		CASE etDiagExtModuleController OF
			TPL.ET_DiagExt.DeactivatingSubModules : 
				stMachineInterface.q_udiDiagExt	:= ET_DiagExt.DeactivatingSubModules;
				stMachineInterface.q_sDiagExt		:= FC_EtDiagExtToString(i_etDiagExt := ET_DiagExt.DeactivatingSubModules);
			TPL.ET_DiagExt.Disabled : 
				stMachineInterface.q_udiDiagExt	:= ET_DiagExt.Disabled;
				stMachineInterface.q_sDiagExt		:= FC_EtDiagExtToString(i_etDiagExt := ET_DiagExt.Disabled);
			TPL.ET_DiagExt.ExecuteStep : 
				stMachineInterface.q_udiDiagExt	:= ET_DiagExt.ExecuteStep;
				stMachineInterface.q_sDiagExt		:= FC_EtDiagExtToString(i_etDiagExt := ET_DiagExt.ExecuteStep);
			TPL.ET_DiagExt.Initializing : 
				stMachineInterface.q_udiDiagExt	:= ET_DiagExt.Initializing;
				stMachineInterface.q_sDiagExt		:= FC_EtDiagExtToString(i_etDiagExt := ET_DiagExt.Initializing);
			TPL.ET_DiagExt.WaitAtNegativeStep : 
				stMachineInterface.q_udiDiagExt	:= ET_DiagExt.WaitAtNegativeStep;
				stMachineInterface.q_sDiagExt		:= FC_EtDiagExtToString(i_etDiagExt := ET_DiagExt.WaitAtNegativeStep);
			TPL.ET_DiagExt.WaitCmdsDone : 
				stMachineInterface.q_udiDiagExt	:= ET_DiagExt.WaitCmdsDone;
				stMachineInterface.q_sDiagExt		:= FC_EtDiagExtToString(i_etDiagExt := ET_DiagExt.WaitCmdsDone);
			TPL.ET_DiagExt.WaitForCmd : 
				stMachineInterface.q_udiDiagExt	:= ET_DiagExt.WaitForCmd;
				stMachineInterface.q_sDiagExt		:= FC_EtDiagExtToString(i_etDiagExt := ET_DiagExt.WaitForCmd);
			ELSE
				stMachineInterface.q_etDiag		:= GD. ET_Diag.UnexpectedProgramBehavior;
				stMachineInterface.q_udiDiagExt	:= ET_DiagExt.UnknownStateModuleController;
				stMachineInterface.q_sDiagExt		:= FC_EtDiagExtToString(i_etDiagExt := ET_DiagExt.UnknownStateModuleController);
		END_CASE
	ELSE
		stMachineInterface.q_etDiag		:= GD.ET_Diag.DiagActive;
		stMachineInterface.q_udiDiagExt	:= ET_DiagExt.ModuleControllerException;
		stMachineInterface.q_sDiagExt		:= FC_EtDiagExtToString(i_etDiagExt := ET_DiagExt.ModuleControllerException);
		stMachineInterface.q_sMsg			:= PDL.FC_MultiConcat(	i_sString1 := GD.FC_EtDiagToString(i_etDiag := etDiagModuleController), 
																			i_sString2 := ' - ',
																			i_sString3 := TPL.FC_EtDiagExtToString(i_etDiagExt := etDiagExtModuleController), 
																			i_sString4 := '');
	END_IF
END_IF
(* End of system generated code, only to be changed by experienced programmers *)
END_ACTION

ACTION PrepStep_Action:
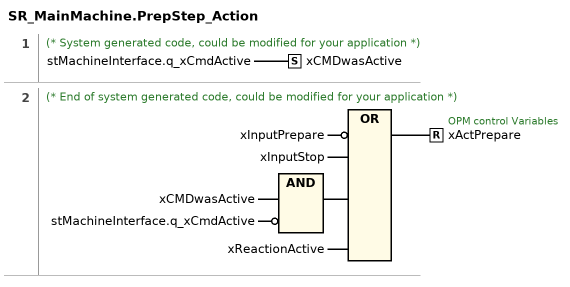
// NETWORK 1
// (* System generated code, could be modified for your application *)
xCMDwasActive S= stMachineInterface.q_xCmdActive;

// NETWORK 2
// (* End of system generated code, could be modified for your application *)
//   xActPrepare: OPM control Variables
xActPrepare R= NOT xInputPrepare OR xInputStop OR xCMDwasActive AND NOT stMachineInterface.q_xCmdActive OR xReactionActive;
END_ACTION

ACTION PrepStep_Entry:
(* System generated code, could be modified for your application *)
	xCMDwasActive:=FALSE;
	stMachineInterface.iq_diCmd	:= ET_Cmd.Prepare;
(* End of system generated code, could be modified for your application *)
END_ACTION

ACTION PrepStop_Action:
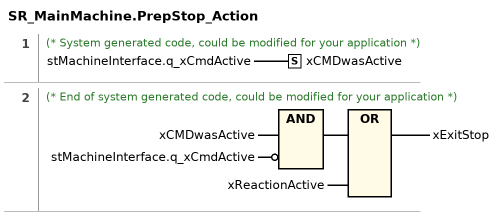
// NETWORK 1
// (* System generated code, could be modified for your application *)
xCMDwasActive S= stMachineInterface.q_xCmdActive;

// NETWORK 2
// (* End of system generated code, could be modified for your application *)
xExitStop := xCMDwasActive AND NOT stMachineInterface.q_xCmdActive OR xReactionActive;
END_ACTION

ACTION PrepStop_Entry:
(* System generated code, could be modified for your application *)
	xCMDwasActive:=FALSE;
	IF	xReactionActive	THEN
		;
	ELSIF stMachineInterface.q_xCmdDone AND NOT stMachineInterface.q_xCmdActive THEN
		stMachineInterface.iq_diCmd	:= ET_Cmd.Stop;
	ELSE
		stMachineInterface.iq_diCmd	:= ET_Cmd.Abort;
	END_IF
(* End of system generated code, could be modified for your application *)
END_ACTION

ACTION StopBrake_Action:
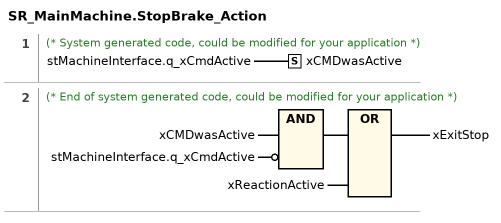
// NETWORK 1
// (* System generated code, could be modified for your application *)
xCMDwasActive S= stMachineInterface.q_xCmdActive;

// NETWORK 2
// (* End of system generated code, could be modified for your application *)
xExitStop := xCMDwasActive AND NOT stMachineInterface.q_xCmdActive OR xReactionActive;
END_ACTION

ACTION StopBrake_Entry:
(* System generated code, could be modified for your application *)
	xCMDwasActive:=FALSE;
	IF	xReactionActive	THEN
		stMachineInterface.iq_diCmd	:= ET_Cmd.Stop;
	ELSIF stMachineInterface.q_xCmdDone AND NOT stMachineInterface.q_xCmdActive THEN
		stMachineInterface.iq_diCmd	:= ET_Cmd.Stop;
	ELSE
		stMachineInterface.iq_diCmd	:= ET_Cmd.Abort;
	END_IF
(* End of system generated code, could be modified for your application *)
END_ACTION

ACTION StopJog_Action:
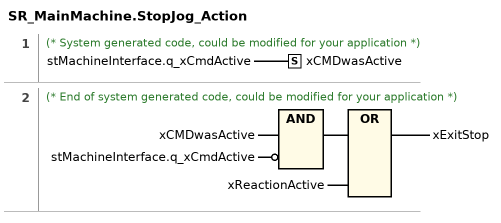
// NETWORK 1
// (* System generated code, could be modified for your application *)
xCMDwasActive S= stMachineInterface.q_xCmdActive;

// NETWORK 2
// (* End of system generated code, could be modified for your application *)
xExitStop := xCMDwasActive AND NOT stMachineInterface.q_xCmdActive OR xReactionActive;
END_ACTION

ACTION StopJog_Entry:
(* System generated code, could be modified for your application *)
	xCMDwasActive:=FALSE;
	IF	xReactionActive	THEN
		;
	ELSIF stMachineInterface.q_xCmdDone AND NOT stMachineInterface.q_xCmdActive THEN
		stMachineInterface.iq_diCmd	:= ET_Cmd.HoldJM;
	ELSE
		stMachineInterface.iq_diCmd	:= ET_Cmd.Abort;
	END_IF
(* End of system generated code, could be modified for your application *)
END_ACTION

ACTION StopMan_Action:
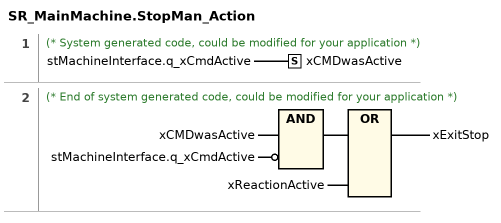
// NETWORK 1
// (* System generated code, could be modified for your application *)
xCMDwasActive S= stMachineInterface.q_xCmdActive;

// NETWORK 2
// (* End of system generated code, could be modified for your application *)
xExitStop := xCMDwasActive AND NOT stMachineInterface.q_xCmdActive OR xReactionActive;
END_ACTION

ACTION StopMan_Entry:
(* System generated code, could be modified for your application *)
	xCMDwasActive:=FALSE;
	IF	xReactionActive	THEN
		;
	ELSIF stMachineInterface.q_xCmdDone AND NOT stMachineInterface.q_xCmdActive THEN
		stMachineInterface.iq_diCmd	:= ET_Cmd.Stop;
	ELSE
		stMachineInterface.iq_diCmd	:= ET_Cmd.Abort;
	END_IF
(* End of system generated code, could be modified for your application *)
END_ACTION

ACTION SubModules_Action:
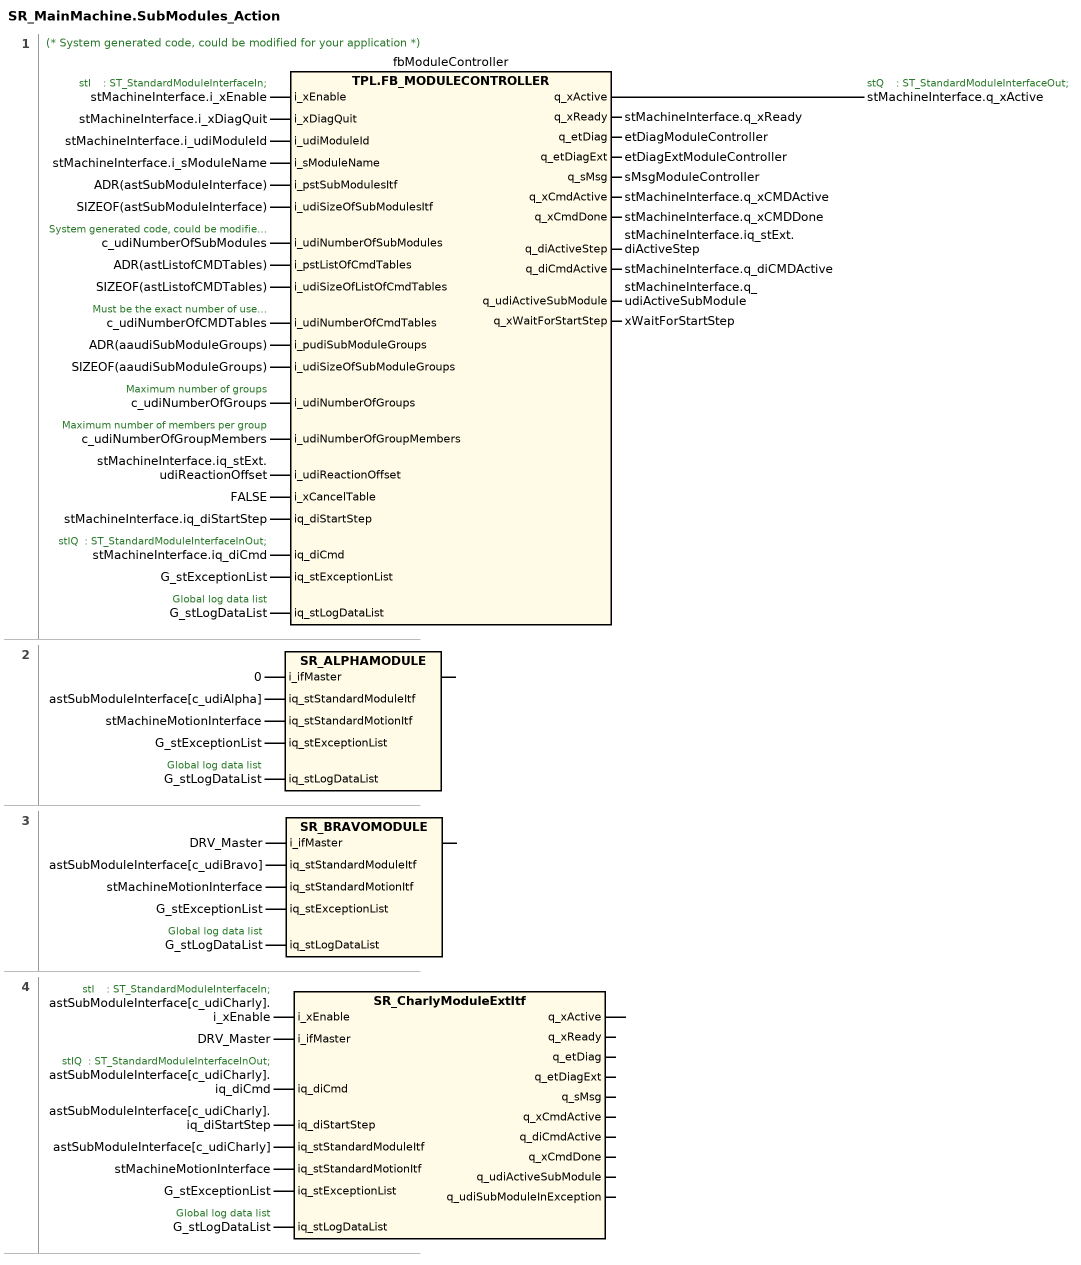
// NETWORK 1
// (* System generated code, could be modified for your application *)
//   fbModuleController: Main ModuleController
//   stMachineInterface.i_xEnable: stI : ST_StandardModuleInterfaceIn;
//   c_udiNumberOfSubModules: System generated code, could be modified for your application
//   c_udiNumberOfCMDTables: Must be the exact number of used CMDTables!
//   c_udiNumberOfGroups: Maximum number of groups
//   c_udiNumberOfGroupMembers: Maximum number of members per group
//   stMachineInterface.iq_diCmd: stIQ : ST_StandardModuleInterfaceInOut;
//   G_stLogDataList: Global log data list
//   stMachineInterface.q_xActive: stQ : ST_StandardModuleInterfaceOut;
fbModuleController(
    i_xEnable := stMachineInterface.i_xEnable,
    i_xDiagQuit := stMachineInterface.i_xDiagQuit,
    i_udiModuleId := stMachineInterface.i_udiModuleId,
    i_sModuleName := stMachineInterface.i_sModuleName,
    i_pstSubModulesItf := ADR(astSubModuleInterface),
    i_udiSizeOfSubModulesItf := SIZEOF(astSubModuleInterface),
    i_udiNumberOfSubModules := c_udiNumberOfSubModules,
    i_pstListOfCmdTables := ADR(astListofCMDTables),
    i_udiSizeOfListOfCmdTables := SIZEOF(astListofCMDTables),
    i_udiNumberOfCmdTables := c_udiNumberOfCMDTables,
    i_pudiSubModuleGroups := ADR(aaudiSubModuleGroups),
    i_udiSizeOfSubModuleGroups := SIZEOF(aaudiSubModuleGroups),
    i_udiNumberOfGroups := c_udiNumberOfGroups,
    i_udiNumberOfGroupMembers := c_udiNumberOfGroupMembers,
    i_udiReactionOffset := stMachineInterface.iq_stExt.udiReactionOffset,
    i_xCancelTable := FALSE,
    iq_diStartStep := stMachineInterface.iq_diStartStep,
    iq_diCmd := stMachineInterface.iq_diCmd,
    iq_stExceptionList := G_stExceptionList,
    iq_stLogDataList := G_stLogDataList,
    q_xReady => stMachineInterface.q_xReady,
    q_etDiag => etDiagModuleController,
    q_etDiagExt => etDiagExtModuleController,
    q_sMsg => sMsgModuleController,
    q_xCmdActive => stMachineInterface.q_xCMDActive,
    q_xCmdDone => stMachineInterface.q_xCMDDone,
    q_diActiveStep => stMachineInterface.iq_stExt.diActiveStep,
    q_diCmdActive => stMachineInterface.q_diCMDActive,
    q_udiActiveSubModule => stMachineInterface.q_udiActiveSubModule,
    q_xWaitForStartStep => xWaitForStartStep); // TPL.FB_MODULECONTROLLER
stMachineInterface.q_xActive := fbModuleController.q_xActive;

// NETWORK 2
//   G_stLogDataList: Global log data list
SR_ALPHAMODULE(i_ifMaster := 0, iq_stStandardModuleItf := astSubModuleInterface[c_udiAlpha], iq_stStandardMotionItf := stMachineMotionInterface, iq_stExceptionList := G_stExceptionList, iq_stLogDataList := G_stLogDataList);

// NETWORK 3
//   G_stLogDataList: Global log data list
SR_BRAVOMODULE(i_ifMaster := DRV_Master, iq_stStandardModuleItf := astSubModuleInterface[c_udiBravo], iq_stStandardMotionItf := stMachineMotionInterface, iq_stExceptionList := G_stExceptionList, iq_stLogDataList := G_stLogDataList);

// NETWORK 4
//   astSubModuleInterface[c_udiCharly].i_xEnable: stI : ST_StandardModuleInterfaceIn;
//   astSubModuleInterface[c_udiCharly].iq_diCmd: stIQ : ST_StandardModuleInterfaceInOut;
//   G_stLogDataList: Global log data list
SR_CharlyModuleExtItf(i_xEnable := astSubModuleInterface[c_udiCharly].i_xEnable, i_ifMaster := DRV_Master, iq_diCmd := astSubModuleInterface[c_udiCharly].iq_diCmd, iq_diStartStep := astSubModuleInterface[c_udiCharly].iq_diStartStep, iq_stStandardModuleItf := astSubModuleInterface[c_udiCharly], iq_stStandardMotionItf := stMachineMotionInterface, iq_stExceptionList := G_stExceptionList, iq_stLogDataList := G_stLogDataList);

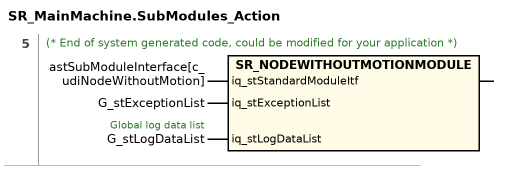
// NETWORK 5
// (* End of system generated code, could be modified for your application *)
//   G_stLogDataList: Global log data list
SR_NODEWITHOUTMOTIONMODULE(iq_stStandardModuleItf := astSubModuleInterface[c_udiNodeWithoutMotion], iq_stExceptionList := G_stExceptionList, iq_stLogDataList := G_stLogDataList);
END_ACTION

ACTION UpdateStructs:
(* System generated code, do not change without consulting 'Schneider Electric Automation GmbH' - otherwise you risk instability!!!*)
fbDetectOnlineChange(	i_xEnable	:= TRUE, 
						i_xDetect	:= TRUE, 
						q_xActive	=> xDetectOnlineChangeActive, 
						q_xReady	=> xDetectOnlineChangeReady, 
						q_etDiag	=> etDetectOnlineChangeDiag, 
						q_etDiagExt	=> etDetectOnlineChangeDiagExt, 
						q_sMsg		=> sDetectOnlineChangeMsg, 
						q_xChange	=> );
						
IF(NOT fbDetectOnlineChange.q_xChange) THEN
	RETURN;
END_IF

stMachineInterface.iq_stExt.udiNumberOfSubModules 		:= c_udiNumberOfSubModules;
stMachineInterface.iq_stExt.dwSubModulesItf		 		:= ADR(astSubModuleInterface);
stMachineInterface.iq_stExt.pdwSubModulesAddItf			:= ADR(adwSubModuleAddInterfaces);
stMachineInterface.iq_stExt.pstListofCMDTables			:= ADR(astListOfCMDTables);
stMachineInterface.iq_stExt.udiNumberOfCmdTables		:= c_udiNumberOfCMDTables;
(* End of system generated code, do not change without consulting 'Schneider Electric Automation GmbH' - otherwise you risk instability!!!*)

(* System generated code, could be modified for your application *)

xUpdateStructsException := FALSE;

(*****************************************************************************************************************************************************)
(* Update CmdTable - Prepare *)

TPL.FC_UpdateCmdTableListElement(	i_pstListofCMDTables	:= ADR(astListofCMDTables),
									i_udiNumberOfCmdTables	:= c_udiNumberOfCMDTables,
									i_diCMD					:= ET_Cmd.Prepare,
									i_pstCMDTable			:= ADR(astPrepareTable),
									q_etDiag				=> etDiag,
									q_etDiagExt				=> etDiagExtTPL);
									
IF etDiag <> GD.ET_Diag.Ok AND NOT xUpdateStructsException THEN
	xUpdateStructsException := TRUE;
	
	stUpdateStructsException.sMsg := PDL.FC_MultiConcat(i_sString1 := 'Update CmdTable: Prepare - ', 
														i_sString2 := GD.FC_EtDiagToString(i_etDiag := etDiag), 
														i_sString3 := ' - ', 
														i_sString4 := TPL.FC_EtDiagExtToString(i_etDiagExt := etDiagExtTPL));
END_IF										

(*****************************************************************************************************************************************************)
(* Update CmdTable - Auto *)

TPL.FC_UpdateCmdTableListElement(	i_pstListofCMDTables	:= ADR(astListofCMDTables),
									i_udiNumberOfCMDTables	:= c_udiNumberOfCMDTables,
									i_diCMD					:= ET_Cmd.Auto,
									i_pstCMDTable			:= ADR(astAutoTable),
									q_etDiag				=> etDiag,
									q_etDiagExt				=> etDiagExtTPL);
									
IF etDiag <> GD.ET_Diag.Ok AND NOT xUpdateStructsException THEN
	xUpdateStructsException := TRUE;
	
	stUpdateStructsException.sMsg := PDL.FC_MultiConcat(i_sString1 := 'Update CmdTable: Auto - ', 
														i_sString2 := GD.FC_EtDiagToString(i_etDiag := etDiag), 
														i_sString3 := ' - ', 
														i_sString4 := TPL.FC_EtDiagExtToString(i_etDiagExt := etDiagExtTPL));
END_IF		

(*****************************************************************************************************************************************************)
(* Update CmdTable - Manual *)

TPL.FC_UpdateCmdTableListElement(	i_pstListofCMDTables	:= ADR(astListofCMDTables),
									i_udiNumberOfCMDTables	:= c_udiNumberOfCMDTables,
									i_diCMD					:= ET_Cmd.Manual,
									i_pstCMDTable			:= ADR(astManualTable),
									q_etDiag				=> etDiag,
									q_etDiagExt				=> etDiagExtTPL);
									
IF etDiag <> GD.ET_Diag.Ok AND NOT xUpdateStructsException THEN
	xUpdateStructsException := TRUE;
	
	stUpdateStructsException.sMsg := PDL.FC_MultiConcat(i_sString1 := 'Update CmdTable: Manual - ', 
														i_sString2 := GD.FC_EtDiagToString(i_etDiag := etDiag), 
														i_sString3 := ' - ', 
														i_sString4 := TPL.FC_EtDiagExtToString(i_etDiagExt := etDiagExtTPL));
END_IF		

(*****************************************************************************************************************************************************)
(* Update CmdTable - Stop *)

TPL.FC_UpdateCmdTableListElement(	i_pstListofCMDTables	:= ADR(astListofCMDTables),
									i_udiNumberOfCMDTables	:= c_udiNumberOfCMDTables,
									i_diCMD					:= ET_Cmd.Stop,
									i_pstCMDTable			:= ADR(astStopTable),
									q_etDiag				=> etDiag,
									q_etDiagExt				=> etDiagExtTPL);
									
IF etDiag <> GD.ET_Diag.Ok AND NOT xUpdateStructsException THEN
	xUpdateStructsException := TRUE;
	
	stUpdateStructsException.sMsg := PDL.FC_MultiConcat(i_sString1 := 'Update CmdTable: Stop - ', 
														i_sString2 := GD.FC_EtDiagToString(i_etDiag := etDiag), 
														i_sString3 := ' - ', 
														i_sString4 := TPL.FC_EtDiagExtToString(i_etDiagExt := etDiagExtTPL));
END_IF		

(*****************************************************************************************************************************************************)
(* Update CmdTable - Start *)

TPL.FC_UpdateCmdTableListElement(	i_pstListofCMDTables	:= ADR(astListofCMDTables),
									i_udiNumberOfCMDTables	:= c_udiNumberOfCMDTables,
									i_diCMD					:= ET_Cmd.Start,
									i_pstCMDTable			:= ADR(astStartTable),
									q_etDiag				=> etDiag,
									q_etDiagExt				=> etDiagExtTPL);
									
IF etDiag <> GD.ET_Diag.Ok AND NOT xUpdateStructsException THEN
	xUpdateStructsException := TRUE;
	
	stUpdateStructsException.sMsg := PDL.FC_MultiConcat(i_sString1 := 'Update CmdTable: Start - ', 
														i_sString2 := GD.FC_EtDiagToString(i_etDiag := etDiag), 
														i_sString3 := ' - ', 
														i_sString4 := TPL.FC_EtDiagExtToString(i_etDiagExt := etDiagExtTPL));
END_IF		

(*****************************************************************************************************************************************************)
(* Update CmdTable - Abort *)

TPL.FC_UpdateCmdTableListElement(	i_pstListofCMDTables	:= ADR(astListofCMDTables),
									i_udiNumberOfCMDTables	:= c_udiNumberOfCMDTables,
									i_diCMD					:= ET_Cmd.Abort,
									i_pstCMDTable			:= ADR(astAbortTable),
									q_etDiag				=> etDiag,
									q_etDiagExt				=> etDiagExtTPL);
									
IF etDiag <> GD.ET_Diag.Ok AND NOT xUpdateStructsException THEN
	xUpdateStructsException := TRUE;
	
	stUpdateStructsException.sMsg := PDL.FC_MultiConcat(i_sString1 := 'Update CmdTable: Abort - ', 
														i_sString2 := GD.FC_EtDiagToString(i_etDiag := etDiag), 
														i_sString3 := ' - ', 
														i_sString4 := TPL.FC_EtDiagExtToString(i_etDiagExt := etDiagExtTPL));
END_IF		

(*****************************************************************************************************************************************************)
(* Update CmdTable - Hold *)

TPL.FC_UpdateCmdTableListElement(	i_pstListofCMDTables	:= ADR(astListofCMDTables),
									i_udiNumberOfCMDTables	:= c_udiNumberOfCMDTables,
									i_diCMD					:= ET_Cmd.Hold,
									i_pstCMDTable			:= ADR(astHoldTable),
									q_etDiag				=> etDiag,
									q_etDiagExt				=> etDiagExtTPL);
									
IF etDiag <> GD.ET_Diag.Ok AND NOT xUpdateStructsException THEN
	xUpdateStructsException := TRUE;
	
	stUpdateStructsException.sMsg := PDL.FC_MultiConcat(i_sString1 := 'Update CmdTable: Hold - ', 
														i_sString2 := GD.FC_EtDiagToString(i_etDiag := etDiag), 
														i_sString3 := ' - ', 
														i_sString4 := TPL.FC_EtDiagExtToString(i_etDiagExt := etDiagExtTPL));
END_IF		

(*****************************************************************************************************************************************************)
(* Update CmdTable - BrakeRelease *)

TPL.FC_UpdateCmdTableListElement(	i_pstListofCMDTables	:= ADR(astListofCMDTables),
									i_udiNumberOfCMDTables	:= c_udiNumberOfCMDTables,
									i_diCMD					:= ET_Cmd.HoldJM,
									i_pstCMDTable			:= ADR(astHoldJogMachineTable),
									q_etDiag				=> etDiag,
									q_etDiagExt				=> etDiagExtTPL);
									
IF etDiag <> GD.ET_Diag.Ok AND NOT xUpdateStructsException THEN
	xUpdateStructsException := TRUE;
	
	stUpdateStructsException.sMsg := PDL.FC_MultiConcat(i_sString1 := 'Update CmdTable: HoldJogMachine - ', 
														i_sString2 := GD.FC_EtDiagToString(i_etDiag := etDiag), 
														i_sString3 := ' - ', 
														i_sString4 := TPL.FC_EtDiagExtToString(i_etDiagExt := etDiagExtTPL));
END_IF		
									
(*****************************************************************************************************************************************************)
(* Update AddInterface - BrakeRelease *)

TPL.FC_UpdateCmdTableListElement(	i_pstListofCMDTables	:= ADR(astListofCMDTables),
									i_udiNumberOfCMDTables	:= c_udiNumberOfCMDTables,
									i_diCMD					:= ET_Cmd.BrakeRelease,
									i_pstCMDTable			:= ADR(astBrakeReleaseTable),
									q_etDiag				=> etDiag,
									q_etDiagExt				=> etDiagExtTPL);
									
IF etDiag <> GD.ET_Diag.Ok AND NOT xUpdateStructsException THEN
	xUpdateStructsException := TRUE;
	
	stUpdateStructsException.sMsg := PDL.FC_MultiConcat(i_sString1 := 'Update CmdTable: BrakeRelease - ', 
														i_sString2 := GD.FC_EtDiagToString(i_etDiag := etDiag), 
														i_sString3 := ' - ', 
														i_sString4 := TPL.FC_EtDiagExtToString(i_etDiagExt := etDiagExtTPL));
END_IF		
									
(*****************************************************************************************************************************************************)
(* Update AddInterface - Jogging *)

TPL.FC_UpdateCmdTableListElement(	i_pstListofCMDTables	:= ADR(astListofCMDTables),
									i_udiNumberOfCMDTables	:= c_udiNumberOfCMDTables,
									i_diCMD					:= ET_Cmd.Jogging,
									i_pstCMDTable			:= ADR(astJogMachineTable),
									q_etDiag				=> etDiag,
									q_etDiagExt				=> etDiagExtTPL);
									
IF etDiag <> GD.ET_Diag.Ok AND NOT xUpdateStructsException THEN
	xUpdateStructsException := TRUE;
	
	stUpdateStructsException.sMsg := PDL.FC_MultiConcat(i_sString1 := 'Update CmdTable: Jogging - ', 
														i_sString2 := GD.FC_EtDiagToString(i_etDiag := etDiag), 
														i_sString3 := ' - ', 
														i_sString4 := TPL.FC_EtDiagExtToString(i_etDiagExt := etDiagExtTPL));
END_IF		
									
(*****************************************************************************************************************************************************)
(* Update AddInterface - Alpha *)

TPL.FC_UpdateNodeModuleAddInterfaceStruct(	i_pdwSubModulesAddItf		:= ADR(adwSubModuleAddInterfaces),
											i_udiSubModuleConstant		:= c_udiAlpha,
											q_etDiag					=> etDiag,
											q_etDiagExt					=> etDiagExtTPL);
									
IF etDiag <> GD.ET_Diag.Ok AND NOT xUpdateStructsException THEN
	xUpdateStructsException := TRUE;
	
	stUpdateStructsException.sMsg := PDL.FC_MultiConcat(i_sString1 := 'Update AddInterface: Alpha - ', 
														i_sString2 := GD.FC_EtDiagToString(i_etDiag := etDiag), 
														i_sString3 := ' - ', 
														i_sString4 := FC_EtDiagExtToString(i_etDiagExt := etDiagExt));
END_IF		
									
(*****************************************************************************************************************************************************)
(* Update AddInterface - Bravo *)

TPL.FC_UpdateNodeModuleAddInterfaceStruct(	i_pdwSubModulesAddItf		:= ADR(adwSubModuleAddInterfaces),
											i_udiSubModuleConstant		:= c_udiBravo,
											q_etDiag					=> etDiag,
											q_etDiagExt					=> etDiagExtTPL);
									
IF etDiag <> GD.ET_Diag.Ok AND NOT xUpdateStructsException THEN
	xUpdateStructsException := TRUE;
	
	stUpdateStructsException.sMsg := PDL.FC_MultiConcat(i_sString1 := 'Update AddInterface: Bravo - ', 
														i_sString2 := GD.FC_EtDiagToString(i_etDiag := etDiag), 
														i_sString3 := ' - ', 
														i_sString4 := FC_EtDiagExtToString(i_etDiagExt := etDiagExt));
END_IF		
									
(*****************************************************************************************************************************************************)
(* Update AddInterface - Charly *)

TPL.FC_UpdateNodeModuleAddInterfaceStruct(	i_pdwSubModulesAddItf		:= ADR(adwSubModuleAddInterfaces),
											i_udiSubModuleConstant		:= c_udiCharly,
											q_etDiag					=> etDiag,
											q_etDiagExt					=> etDiagExtTPL);
									
IF etDiag <> GD.ET_Diag.Ok AND NOT xUpdateStructsException THEN
	xUpdateStructsException := TRUE;
	
	stUpdateStructsException.sMsg := PDL.FC_MultiConcat(i_sString1 := 'Update AddInterface: Charly - ', 
														i_sString2 := GD.FC_EtDiagToString(i_etDiag := etDiag), 
														i_sString3 := ' - ', 
														i_sString4 := FC_EtDiagExtToString(i_etDiagExt := etDiagExt));
END_IF		
									
(*****************************************************************************************************************************************************)
(* Update AddInterface - NodeWithoutMotion *)

TPL.FC_UpdateNodeModuleAddInterfaceStruct(	i_pdwSubModulesAddItf		:= ADR(adwSubModuleAddInterfaces),
											i_udiSubModuleConstant		:= c_udiNodeWithoutMotion,
											q_etDiag					=> etDiag,
											q_etDiagExt					=> etDiagExtTPL);
									
IF etDiag <> GD.ET_Diag.Ok AND NOT xUpdateStructsException THEN
	xUpdateStructsException := TRUE;
	
	stUpdateStructsException.sMsg := PDL.FC_MultiConcat(i_sString1 := 'Update AddInterface: NodeWithoutMotion - ', 
														i_sString2 := GD.FC_EtDiagToString(i_etDiag := etDiag), 
														i_sString3 := ' - ', 
														i_sString4 := FC_EtDiagExtToString(i_etDiagExt := etDiagExt));
END_IF		

(*****************************************************************************************************************************************************)
(* Set exception if any exception occurred *)

TPL.FC_SetException(i_xExceptionActive	:= xUpdateStructsException, 
					iq_stException		:= stUpdateStructsException, 
					iq_stExceptionList	:= G_stExceptionList, 
					iq_stLogDataList	:= G_stLogDataList);
					
xInitSuccessful := xInitSuccessful AND NOT xUpdateStructsException;

etDiag := GD.ET_Diag.Ok;

(* End of system generated code, could be modified for your application *)
END_ACTION

END_PROGRAM

// LMC_PacDrive/Application/CrankModuleExample/ProjectDiagnostics/FC_EtDiagExtToString
FUNCTION FC_EtDiagExtToString : STRING[80]

VAR_INPUT
	i_etDiagExt : ET_DiagExt;
END_VAR

VAR_OUTPUT
	q_etDiag	: GD.ET_Diag := GD.ET_Diag.Ok;
	q_etDiagExt	: ET_DiagExt := ET_DiagExt.Ok;
END_VAR

VAR
END_VAR

CASE i_etDiagExt OF
	ET_DiagExt.Ok:								FC_EtDiagExtToString := 'Ok';
	ET_DiagExt.Disabled:						FC_EtDiagExtToString := 'Disabled';
	ET_DiagExt.WaitUntilControllerFinishedBoot:	FC_EtDiagExtToString := 'WaitUntilControllerFinishedBoot';
	ET_DiagExt.Initializing:					FC_EtDiagExtToString := 'Initializing';
	ET_DiagExt.DeactivatingSubModules:			FC_EtDiagExtToString := 'DeactivatingSubModules';
	ET_DiagExt.ExecuteStep:						FC_EtDiagExtToString := 'ExecuteStep';
	ET_DiagExt.WaitAtNegativeStep:				FC_EtDiagExtToString := 'WaitAtNegativeStep';
	ET_DiagExt.WaitCmdsDone:					FC_EtDiagExtToString := 'WaitCmdsDone';
	ET_DiagExt.WaitForCmd:						FC_EtDiagExtToString := 'WaitForCmd';
	ET_DiagExt.SubModuleInException:			FC_EtDiagExtToString := 'SubModuleInException';
	ET_DiagExt.ModuleControllerException:		FC_EtDiagExtToString := 'ModuleControllerException';
	ET_DiagExt.UnknownStateModuleController:	FC_EtDiagExtToString := 'UnknownStateModuleController';
	
	ET_DiagExt.SystemFatalException:			FC_EtDiagExtToString := 'SystemFatalException';
	ET_DiagExt.SystemException:					FC_EtDiagExtToString := 'SystemException';
	ET_DiagExt.SystemWarning:					FC_EtDiagExtToString := 'SystemWarning';
	ET_DiagExt.MainSystemEmergencyStop:			FC_EtDiagExtToString := 'MainSystemEmergencyStop';
	ET_DiagExt.InvalidPointer:					FC_EtDiagExtToString := 'InvalidPointer';
	ET_DiagExt.UpdateStructsException:			FC_EtDiagExtToString := 'UpdateStructsException';
	ET_DiagExt.InitReactionsException:			FC_EtDiagExtToString := 'InitReactionsException';
	ET_DiagExt.InitSubModulesException:			FC_EtDiagExtToString := 'InitSubModulesException';
	ET_DiagExt.DriveInvalid:					FC_EtDiagExtToString := 'DriveInvalid';
	ET_DiagExt.UnknownDiagExt:					FC_EtDiagExtToString := 'UnknownDiagExt';

	ET_DiagExt.Exception1FromVis:				FC_EtDiagExtToString := 'Exception1FromVis';
	ET_DiagExt.Exception2FromVis:				FC_EtDiagExtToString := 'Exception2FromVis';
	ET_DiagExt.Exception3FromVis:				FC_EtDiagExtToString := 'Exception3FromVis';
	ET_DiagExt.Exception4FromVis:				FC_EtDiagExtToString := 'Exception4FromVis';
	ET_DiagExt.Exception5FromVis:				FC_EtDiagExtToString := 'Exception5FromVis';
	
	ET_DiagExt.DiagnosticsWarning:				FC_EtDiagExtToString := 'DiagnosticsWarning';
	ET_DiagExt.WaitUntilDiagnosticsManagerReady:FC_EtDiagExtToString := 'WaitUntilDiagnosticsManagerReady';
	ET_DiagExt.WaitUntilDisabled:				FC_EtDiagExtToString := 'WaitUntilDisabled';
	ET_DiagExt.WaitUntilDiagSourceRegistered:	FC_EtDiagExtToString := 'WaitUntilDiagSourceRegistered';
	ET_DiagExt.WaitForCommunication:			FC_EtDiagExtToString := 'WaitForCommunication';
	ET_DiagExt.DataSuccessfullyWritten:			FC_EtDiagExtToString := 'DataSuccessfullyWritten';
	ET_DiagExt.WritingToFile:					FC_EtDiagExtToString := 'WritingToFile';
	ET_DiagExt.FileIdInvalid:					FC_EtDiagExtToString := 'FileIdInvalid';
	ET_DiagExt.CmdUnknown:						FC_EtDiagExtToString := 'CmdUnknown';
	ET_DiagExt.UnexpectedFeedback:				FC_EtDiagExtToString := 'UnexpectedFeedback';
	ET_DiagExt.UnknownDiagExtUser:				FC_EtDiagExtToString := 'UnknownDiagExtUser';
ELSE
	FC_EtDiagExtToString := CONCAT('Unkown ET_DiagExt ', UDINT_TO_STRING(i_etDiagExt));
		
	q_etDiag	:= GD.ET_Diag.InputParameterInvalid;
	q_etDiagExt	:= ET_DiagExt.UnknownDiagExt;
END_CASE

END_FUNCTION

// LMC_PacDrive/Application/CrankModuleExample/ProjectDiagnostics/FC_EtDiagExtUserToString
FUNCTION FC_EtDiagExtUserToString : STRING[80]
VAR_INPUT
	i_etDiagExt : ET_DiagExtUser;
END_VAR
VAR_OUTPUT
	q_etDiag	: GD.ET_Diag := GD.ET_Diag.Ok;
	q_etDiagExt	: ET_DiagExt := ET_DiagExt.Ok;
END_VAR
VAR
END_VAR

CASE i_etDiagExt OF
	ET_DiagExtUser.Exception1FromEquipmentModule	: FC_EtDiagExtUserToString := 'Exception1FromEquipmentModule';
	ET_DiagExtUser.Exception2FromEquipmentModule	: FC_EtDiagExtUserToString := 'Exception2FromEquipmentModule';
	
	ET_DiagExtUser.Exception1FromMain				: FC_EtDiagExtUserToString := 'Exception1FromMain';
	ET_DiagExtUser.Exception2FromMain				: FC_EtDiagExtUserToString := 'Exception2FromMain';
	ET_DiagExtUser.Exception3FromMain				: FC_EtDiagExtUserToString := 'Exception3FromMain';
	ET_DiagExtUser.Exception4FromMain				: FC_EtDiagExtUserToString := 'Exception4FromMain';
	ET_DiagExtUser.Exception5FromMain				: FC_EtDiagExtUserToString := 'Exception5FromMain';
ELSE
	FC_EtDiagExtUserToString := CONCAT('Unkown ET_DiagExtUser ', UDINT_TO_STRING(i_etDiagExt));
		
	q_etDiag	:= GD.ET_Diag.InputParameterInvalid;
	q_etDiagExt	:= ET_DiagExt.UnknownDiagExtUser;
END_CASE

END_FUNCTION

// LMC_PacDrive/Application/CrankModuleExample/EquipmentModules/SR_AlphaModule
PROGRAM SR_AlphaModule

VAR CONSTANT
(* Standard related constants *)
	c_udiNumberOfGroups				: UDINT := 0;			(* Maximum number of groups *)
	c_udiNumberOfGroupMembers		: UDINT := 0;			(* Maximum number of members per group *)

	c_udiNumberOfCmdTables			: UDINT := 8;			(* Must be the exact number of used CmdTables! *)
	c_udiNumberOfCmdSteps			: UDINT := 16;			(* Make sure that the number of command steps that each table
															   contains does not exceed the c_diNumberOfCmdSteps variable. *)

(* Definition group of modules *)
	c_udiAlphaGroup1				: UDINT := 2001;		(* Name of module group  1 *)
	c_udiAlphaGroup2				: UDINT := 2002;		(* Name of module group  2 *)

(* System generated code, could be modified for your application *)
	c_udiNumberOfSubModules			: UDINT := 1;			(* Number of SubModules *)
	c_udiMaster						: UDINT := 1;
(* End of system generated code, could be modified for your application *)
END_VAR

VAR (* User specific variables *)
	stMasterInterface				: AXM.ST_ModuleInterface;
	fbMasterModule					: AXM.FB_AxisModule;

	fbAxisModuleController			: AXM.FB_AxisModuleController;
END_VAR

VAR_INPUT
(* Master of AlphaModule *)
	i_ifMaster						: SystemConfigurationItf.IF_Master;
END_VAR

VAR_IN_OUT
(* TPL.ST_StandardModuleInterface *)	
	iq_stStandardModuleItf			: TPL.ST_StandardModuleInterface;
	
(* TPL.ST_StandardMotionInterface *)		
	iq_stStandardMotionItf			: TPL.ST_StandardMotionInterface;
	
(* ExceptionHandling and Logging *)	
	iq_stExceptionList				: TPL.ST_ExceptionList;
	iq_stLogDataList				: TPL.ST_LogDataList;
END_VAR

VAR
	xInitSuccessful : BOOL := TRUE;
	
(* Standard related variables *)
	astSubModuleInterface			: ARRAY[1..c_udiNumberOfSubModules] OF TPL.ST_StandardModuleInterface;		(* Interface to modules *)
	aaudiSubModuleGroups			: ARRAY[1..c_udiNumberOfGroups,1..c_udiNumberOfGroupMembers] OF UDINT;
	adwSubModuleAddInterfaces		: ARRAY[1..c_udiNumberOfSubModules] OF DWORD;

(* Modules related variables *)
	fbModuleController				: TPL.FB_ModuleController;
	etDiagModuleController			: GD.ET_Diag;
	etDiagExtModuleController		: TPL.ET_DiagExt;
	sMsgModuleController			: STRING[80];
	xWaitForStartStep				: BOOL;
	
	astListOfCmdTables				: ARRAY [1..c_udiNumberOfCmdTables] OF TPL.ST_CmdTable;
	udiTableIndex					: UDINT;
	udiStepIndex					: UDINT;
	diStep							: DINT;

	astPrepareTable					: ARRAY [1..c_udiNumberOfCmdSteps] OF TPL.ST_Cmd;		(* Relating Cmd table *)
	astAutoTable					: ARRAY [1..c_udiNumberOfCmdSteps] OF TPL.ST_Cmd;		(* Relating Cmd table *)
	astManualTable					: ARRAY [1..c_udiNumberOfCmdSteps] OF TPL.ST_Cmd;		(* Relating Cmd table *)
	astHoldTable					: ARRAY [1..c_udiNumberOfCmdSteps] OF TPL.ST_Cmd;		(* Relating Cmd table *)
	astStartTable					: ARRAY [1..c_udiNumberOfCmdSteps] OF TPL.ST_Cmd;		(* Relating Cmd table *)
	astStopTable					: ARRAY [1..c_udiNumberOfCmdSteps] OF TPL.ST_Cmd;		(* Relating Cmd table *)
	astBrakeReleaseTable			: ARRAY [1..c_udiNumberOfCmdSteps] OF TPL.ST_Cmd;		(* Relating Cmd table *)
	astAbortTable					: ARRAY [1..c_udiNumberOfCmdSteps] OF TPL.ST_Cmd;		(* Relating Cmd table *)

(* ExceptionHandling related variables *)
	fbExceptionHandler				: TPL.FB_ExceptionHandler;

	aetReactionTranslationMode		: ARRAY[1..c_udiNumberOfSubModules] OF TPL.ET_ReactionTranslationMode;
	aastReactionTranslationTable	: ARRAY[1..c_udiNumberOfSubModules,1..TPL.Gc_udiMaxNumberOfReactions] OF TPL.ST_Reaction;
	astReactionTranslationJobs		: ARRAY[1..c_udiNumberOfSubModules] OF TPL.ST_ReactionTranslationJobs;

(* Exception declaration *)
	stUserException1				: TPL.ST_Exception;
	stUserException2				: TPL.ST_Exception;
	xModuleUserException1			: BOOL;
	xModuleUserException2			: BOOL;
	
	stUpdateStructsException		: TPL.ST_Exception;
	xUpdateStructsException			: BOOL;
	
	stInitReactionsException		: TPL.ST_Exception;
	xInitReactionsException			: BOOL;
	
	stInitSubModulesException		: TPL.ST_Exception;
	xInitSubModulesException		: BOOL;
	
	stIsDriveVirtualException		: TPL.ST_Exception;
	xIsDriveVirtualException		: BOOL;

(* Logging related variables*)
	fbLogger						: TPL.FB_Logger;

(* OnlineChange related variables *)
	fbDetectOnlineChange			: TPL.FB_DetectOnlineChange;
	xDetectOnlineChangeActive		: BOOL; 
	xDetectOnlineChangeReady		: BOOL; 
	etDetectOnlineChangeDiag		: GD.ET_Diag;
	etDetectOnlineChangeDiagExt		: TPL.ET_DiagExt; 
	sDetectOnlineChangeMsg			: STRING[80];
	
(* Init related variables *)	
	stLogicalAddressMaster			: SystemConfigurationItf.ST_LogicalAddress;
	lrShaftRefDelay					: LREAL;
	diResult						: DINT;

	xDriveIsVirtual					: BOOL;	
	
(* POU-Feedback related variables*)	
	etDiag			: GD.ET_Diag;
	etDiagExt		: ET_DiagExt;
	etDiagExtTPL	: TPL.ET_DiagExt;
	etDiagExtAXM	: AXM.ET_DiagExt;
	sMsgBuffer		: STRING[80];
END_VAR

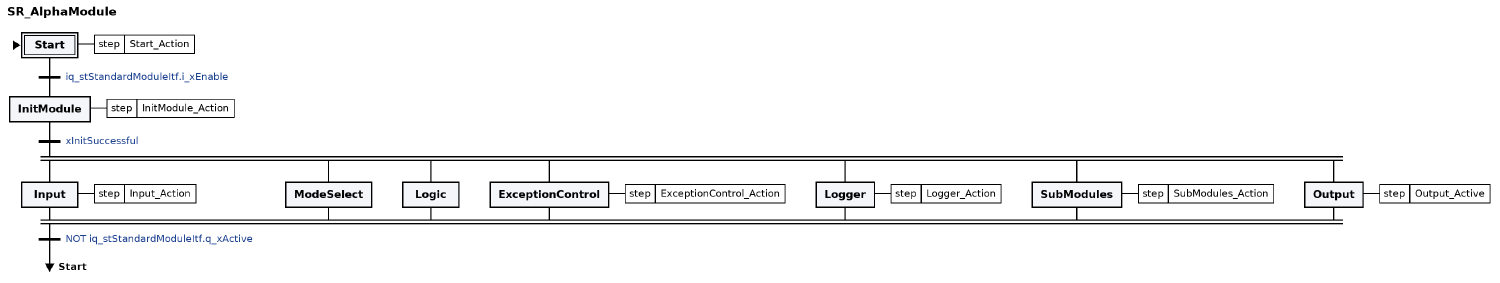
INITIAL_STEP Start:
    Start_Action(N);  // step action
END_STEP
TRANSITION FROM Start TO InitModule
    := iq_stStandardModuleItf.i_xEnable;
END_TRANSITION
STEP InitModule:
    InitModule_Action(N);  // step action
END_STEP
TRANSITION FROM InitModule TO (Input, ModeSelect, Logic, ExceptionControl, Logger, SubModules, Output)
    := xInitSuccessful;
END_TRANSITION
STEP Input:
    Input_Action(N);  // step action
END_STEP
STEP ModeSelect:
END_STEP
STEP Logic:
END_STEP
STEP ExceptionControl:
    ExceptionControl_Action(N);  // step action
END_STEP
STEP Logger:
    Logger_Action(N);  // step action
END_STEP
STEP SubModules:
    SubModules_Action(N);  // step action
END_STEP
STEP Output:
    Output_Active(N);  // step action
END_STEP
TRANSITION FROM (Input, ModeSelect, Logic, ExceptionControl, Logger, SubModules, Output) TO Start
    := NOT iq_stStandardModuleItf.q_xActive;
END_TRANSITION

ACTION ExceptionControl_Action:
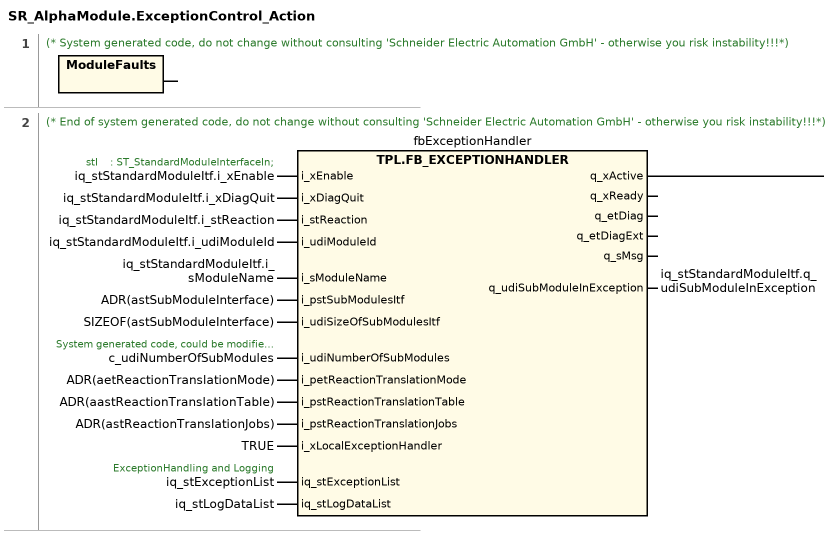
// NETWORK 1
// (* System generated code, do not change without consulting 'Schneider Electric Automation GmbH' - otherwise you risk instability!!!*)
ModuleFaults();

// NETWORK 2
// (* End of system generated code, do not change without consulting 'Schneider Electric Automation GmbH' - otherwise you risk instability!!!*)
//   fbExceptionHandler: ExceptionHandling related variables
//   iq_stStandardModuleItf.i_xEnable: stI : ST_StandardModuleInterfaceIn;
//   c_udiNumberOfSubModules: System generated code, could be modified for your application
//   iq_stExceptionList: ExceptionHandling and Logging
fbExceptionHandler(
    i_xEnable := iq_stStandardModuleItf.i_xEnable,
    i_xDiagQuit := iq_stStandardModuleItf.i_xDiagQuit,
    i_stReaction := iq_stStandardModuleItf.i_stReaction,
    i_udiModuleId := iq_stStandardModuleItf.i_udiModuleId,
    i_sModuleName := iq_stStandardModuleItf.i_sModuleName,
    i_pstSubModulesItf := ADR(astSubModuleInterface),
    i_udiSizeOfSubModulesItf := SIZEOF(astSubModuleInterface),
    i_udiNumberOfSubModules := c_udiNumberOfSubModules,
    i_petReactionTranslationMode := ADR(aetReactionTranslationMode),
    i_pstReactionTranslationTable := ADR(aastReactionTranslationTable),
    i_pstReactionTranslationJobs := ADR(astReactionTranslationJobs),
    i_xLocalExceptionHandler := TRUE,
    iq_stExceptionList := iq_stExceptionList,
    iq_stLogDataList := iq_stLogDataList,
    q_udiSubModuleInException => iq_stStandardModuleItf.q_udiSubModuleInException); // TPL.FB_EXCEPTIONHANDLER
END_ACTION

ACTION Init_CmdTables:
(* System generated code, could be modified for your application *)

(*********************************************************************************************************************)
(*** Prepare  ***)

TPL.FC_FirstStep(udiStepIndex, diStep);
astPrepareTable[udiStepIndex].sTitle					:= 'DriveEnable On AllSubModules';
astPrepareTable[udiStepIndex].udiModuleName				:= TPL.Gc_udiAllSubModules;
astPrepareTable[udiStepIndex].diStep					:= diStep;
astPrepareTable[udiStepIndex].diCMD						:= AXM.ET_Cmd.DriveEnableOn;
astPrepareTable[udiStepIndex].timTimeOut				:= T#0MS;
astPrepareTable[udiStepIndex].xEndCMD					:= FALSE;

TPL.FC_NextStep(udiStepIndex, diStep);
astPrepareTable[udiStepIndex].sTitle					:= 'Homing Mode AllSubModules';
astPrepareTable[udiStepIndex].udiModuleName				:= TPL.Gc_udiAllSubModules;
astPrepareTable[udiStepIndex].diStep					:= diStep;
astPrepareTable[udiStepIndex].diCMD						:= AXM.ET_Cmd.Homing;
astPrepareTable[udiStepIndex].timTimeOut				:= T#0MS;
astPrepareTable[udiStepIndex].xEndCMD					:= FALSE;

TPL.FC_NextStep(udiStepIndex, diStep);
astPrepareTable[udiStepIndex].sTitle					:= 'Start AllSubModules';
astPrepareTable[udiStepIndex].udiModuleName				:= TPL.Gc_udiAllSubModules;
astPrepareTable[udiStepIndex].diStep					:= diStep;
astPrepareTable[udiStepIndex].diCMD						:= AXM.ET_Cmd.Start;
astPrepareTable[udiStepIndex].timTimeOut				:= T#0MS;
astPrepareTable[udiStepIndex].xEndCMD					:= FALSE;

TPL.FC_LastStep(udiStepIndex, diStep);
astPrepareTable[udiStepIndex].sTitle					:= 'End';
astPrepareTable[udiStepIndex].udiModuleName				:= 0;
astPrepareTable[udiStepIndex].diStep					:= diStep;
astPrepareTable[udiStepIndex].diCMD						:= 0;
astPrepareTable[udiStepIndex].timTimeOut				:= T#0MS;
astPrepareTable[udiStepIndex].xEndCMD					:= TRUE;

TPL.FC_FirstCmdTable(iq_udiTableIndex := udiTableIndex);
astListofCMDTables[udiTableIndex].sTitle				:= 'Prepare';
astListofCMDTables[udiTableIndex].diCMD					:= ET_Cmd.Prepare;
astListofCMDTables[udiTableIndex].udiNumberOfCmdSteps	:= udiStepIndex;

(*********************************************************************************************************************)
(*** Auto  ***)

TPL.FC_FirstStep(udiStepIndex, diStep);
astAutoTable[udiStepIndex].sTitle						:= 'DriveEnable On AllSubModules';
astAutoTable[udiStepIndex].udiModuleName				:= TPL.Gc_udiAllSubModules;
astAutoTable[udiStepIndex].diStep						:= diStep;
astAutoTable[udiStepIndex].diCMD						:= AXM.ET_Cmd.DriveEnableOn;
astAutoTable[udiStepIndex].timTimeOut					:= T#0MS;
astAutoTable[udiStepIndex].xEndCMD						:= FALSE;

TPL.FC_NextStep(udiStepIndex, diStep);
astAutoTable[udiStepIndex].sTitle						:= 'Endless Mode AllSubModules';
astAutoTable[udiStepIndex].udiModuleName				:= TPL.Gc_udiAllSubModules;
astAutoTable[udiStepIndex].diStep						:= diStep;
astAutoTable[udiStepIndex].diCMD						:= AXM.ET_Cmd.Endless;
astAutoTable[udiStepIndex].timTimeOut					:= T#0MS;
astAutoTable[udiStepIndex].xEndCMD						:= FALSE;

TPL.FC_NextStep(udiStepIndex, diStep);
astAutoTable[udiStepIndex].sTitle						:= 'Start AllSubModules';
astAutoTable[udiStepIndex].udiModuleName				:= TPL.Gc_udiAllSubModules;
astAutoTable[udiStepIndex].diStep						:= diStep;
astAutoTable[udiStepIndex].diCMD						:= AXM.ET_Cmd.Start;
astAutoTable[udiStepIndex].timTimeOut					:= T#0MS;
astAutoTable[udiStepIndex].xEndCMD						:= FALSE;

TPL.FC_LastStep(udiStepIndex, diStep);
astAutoTable[udiStepIndex].sTitle						:= 'End';
astAutoTable[udiStepIndex].udiModuleName				:= 0;
astAutoTable[udiStepIndex].diStep						:= diStep;
astAutoTable[udiStepIndex].diCMD						:= 0;
astAutoTable[udiStepIndex].timTimeOut					:= T#0MS;
astAutoTable[udiStepIndex].xEndCMD						:= TRUE;

TPL.FC_NextCmdTable(iq_udiTableIndex:= udiTableIndex);
astListofCMDTables[udiTableIndex].sTitle				:= 'Auto';
astListofCMDTables[udiTableIndex].diCMD					:= ET_Cmd.Auto;
astListofCMDTables[udiTableIndex].udiNumberOfCmdSteps	:= udiStepIndex;

(*********************************************************************************************************************)
(*** Manual  ***)

TPL.FC_FirstStep(udiStepIndex, diStep);
astManualTable[udiStepIndex].sTitle						:= 'DriveEnable On AllSubModules';
astManualTable[udiStepIndex].udiModuleName				:= TPL.Gc_udiAllSubModules;
astManualTable[udiStepIndex].diStep						:= diStep;
astManualTable[udiStepIndex].diCMD						:= AXM.ET_Cmd.DriveEnableOn;
astManualTable[udiStepIndex].timTimeOut					:= T#0MS;
astManualTable[udiStepIndex].xEndCMD					:= FALSE;

TPL.FC_NextStep(udiStepIndex, diStep);
astManualTable[udiStepIndex].sTitle						:= 'Manual Mode AllSubModules';
astManualTable[udiStepIndex].udiModuleName				:= TPL.Gc_udiAllSubModules;
astManualTable[udiStepIndex].diStep						:= diStep;
astManualTable[udiStepIndex].diCMD						:= AXM.ET_Cmd.Manual;
astManualTable[udiStepIndex].timTimeOut					:= T#0MS;
astManualTable[udiStepIndex].xEndCMD					:= FALSE;

TPL.FC_LastStep(udiStepIndex, diStep);
astManualTable[udiStepIndex].sTitle						:= 'End';
astManualTable[udiStepIndex].udiModuleName				:= 0;
astManualTable[udiStepIndex].diStep						:= diStep;
astManualTable[udiStepIndex].diCMD						:= 0;
astManualTable[udiStepIndex].timTimeOut					:= T#0MS;
astManualTable[udiStepIndex].xEndCMD					:= TRUE;

TPL.FC_NextCmdTable(iq_udiTableIndex:= udiTableIndex);
astListofCMDTables[udiTableIndex].sTitle				:= 'Manual';
astListofCMDTables[udiTableIndex].diCMD					:= ET_Cmd.Manual;
astListofCMDTables[udiTableIndex].udiNumberOfCmdSteps	:= udiStepIndex;

(*********************************************************************************************************************)
(*** Stop ***)

TPL.FC_FirstStep(udiStepIndex, diStep);
astStopTable[udiStepIndex].sTitle						:= 'Stop AllSubModules';
astStopTable[udiStepIndex].udiModuleName				:= TPL.Gc_udiAllSubModules;
astStopTable[udiStepIndex].diStep						:= diStep;
astStopTable[udiStepIndex].diCMD						:= AXM.ET_Cmd.Stop;
astStopTable[udiStepIndex].timTimeOut					:= T#0MS;
astStopTable[udiStepIndex].xEndCMD						:= FALSE;

TPL.FC_LastStep(udiStepIndex, diStep);
astStopTable[udiStepIndex].sTitle						:= 'End';
astStopTable[udiStepIndex].udiModuleName				:= 0;
astStopTable[udiStepIndex].diStep						:= diStep;
astStopTable[udiStepIndex].diCMD						:= 0;
astStopTable[udiStepIndex].timTimeOut					:= T#0MS;
astStopTable[udiStepIndex].xEndCMD						:= TRUE;

TPL.FC_NextCmdTable(iq_udiTableIndex:= udiTableIndex);
astListofCMDTables[udiTableIndex].sTitle				:= 'Stop';
astListofCMDTables[udiTableIndex].diCMD					:= ET_Cmd.Stop;
astListofCMDTables[udiTableIndex].udiNumberOfCmdSteps	:= udiStepIndex;

(*********************************************************************************************************************)
(*** Start ***)

TPL.FC_FirstStep(udiStepIndex, diStep);
astStartTable[udiStepIndex].sTitle						:= 'Start AllSubModules';
astStartTable[udiStepIndex].udiModuleName				:= TPL.Gc_udiAllSubModules;
astStartTable[udiStepIndex].diStep						:= diStep;
astStartTable[udiStepIndex].diCMD						:= AXM.ET_Cmd.Start;
astStartTable[udiStepIndex].timTimeOut					:= T#0MS;
astStartTable[udiStepIndex].xEndCMD						:= FALSE;

TPL.FC_LastStep(udiStepIndex, diStep);
astStartTable[udiStepIndex].sTitle						:= 'End';
astStartTable[udiStepIndex].udiModuleName				:= 0;
astStartTable[udiStepIndex].diStep						:= diStep;
astStartTable[udiStepIndex].diCMD						:= 0;
astStartTable[udiStepIndex].timTimeOut					:= T#0MS;
astStartTable[udiStepIndex].xEndCMD						:= TRUE;

TPL.FC_NextCmdTable(iq_udiTableIndex:= udiTableIndex);
astListofCMDTables[udiTableIndex].sTitle				:= 'Start';
astListofCMDTables[udiTableIndex].diCMD					:= ET_Cmd.Start;
astListofCMDTables[udiTableIndex].udiNumberOfCmdSteps	:= udiStepIndex;

(*********************************************************************************************************************)
(*** Abort ***)

TPL.FC_FirstStep(udiStepIndex, diStep);
astAbortTable[udiStepIndex].sTitle						:= 'Stop AllSubModules';
astAbortTable[udiStepIndex].udiModuleName				:= TPL.Gc_udiAllSubModules;
astAbortTable[udiStepIndex].diStep						:= diStep;
astAbortTable[udiStepIndex].diCMD						:= AXM.ET_Cmd.Stop;
astAbortTable[udiStepIndex].timTimeOut					:= T#0MS;
astAbortTable[udiStepIndex].xEndCMD						:= FALSE;

TPL.FC_LastStep(udiStepIndex, diStep);
astAbortTable[udiStepIndex].sTitle						:= 'End';
astAbortTable[udiStepIndex].udiModuleName				:= 0;
astAbortTable[udiStepIndex].diStep						:= diStep;
astAbortTable[udiStepIndex].diCMD						:= 0;
astAbortTable[udiStepIndex].timTimeOut					:= T#0MS;
astAbortTable[udiStepIndex].xEndCMD						:= TRUE;

TPL.FC_NextCmdTable(iq_udiTableIndex:= udiTableIndex);
astListofCMDTables[udiTableIndex].sTitle				:= 'Abort';
astListofCMDTables[udiTableIndex].diCMD					:= ET_Cmd.Abort;
astListofCMDTables[udiTableIndex].udiNumberOfCmdSteps	:= udiStepIndex;

(*********************************************************************************************************************)
(*** Hold ***)

TPL.FC_FirstStep(udiStepIndex, diStep);
astHoldTable[udiStepIndex].sTitle						:= 'Hold AllSubModules';
astHoldTable[udiStepIndex].udiModuleName				:= TPL.Gc_udiAllSubModules;
astHoldTable[udiStepIndex].diStep						:= diStep;
astHoldTable[udiStepIndex].diCMD						:= AXM.ET_Cmd.Hold;
astHoldTable[udiStepIndex].timTimeOut					:= T#0MS;
astHoldTable[udiStepIndex].xEndCMD						:= FALSE;

TPL.FC_LastStep(udiStepIndex, diStep);
astHoldTable[udiStepIndex].sTitle						:= 'End';
astHoldTable[udiStepIndex].udiModuleName				:= 0;
astHoldTable[udiStepIndex].diStep						:= diStep;
astHoldTable[udiStepIndex].diCMD						:= 0;
astHoldTable[udiStepIndex].timTimeOut					:= T#0MS;
astHoldTable[udiStepIndex].xEndCMD						:= TRUE;

TPL.FC_NextCmdTable(iq_udiTableIndex:= udiTableIndex);
astListofCMDTables[udiTableIndex].sTitle				:= 'Hold';
astListofCMDTables[udiTableIndex].diCMD					:= ET_Cmd.Hold;
astListofCMDTables[udiTableIndex].udiNumberOfCmdSteps	:= udiStepIndex;

(*********************************************************************************************************************)
(*** Brake Release ***)

TPL.FC_FirstStep(udiStepIndex, diStep);
astBrakeReleaseTable[udiStepIndex].sTitle				:= 'DriveEnable Off AllSubModules';
astBrakeReleaseTable[udiStepIndex].udiModuleName		:= TPL.Gc_udiAllSubModules;
astBrakeReleaseTable[udiStepIndex].diStep				:= diStep;
astBrakeReleaseTable[udiStepIndex].diCMD				:= AXM.ET_Cmd.DriveEnableOff;
astBrakeReleaseTable[udiStepIndex].timTimeOut			:= T#0MS;
astBrakeReleaseTable[udiStepIndex].xEndCMD				:= FALSE;

TPL.FC_NextStep(udiStepIndex, diStep);
astBrakeReleaseTable[udiStepIndex].sTitle				:= 'BrakeRelease Mode AllSubModules';
astBrakeReleaseTable[udiStepIndex].udiModuleName		:= TPL.Gc_udiAllSubModules;
astBrakeReleaseTable[udiStepIndex].diStep				:= diStep;
astBrakeReleaseTable[udiStepIndex].diCMD				:= AXM.ET_Cmd.BrakeRelease;
astBrakeReleaseTable[udiStepIndex].timTimeOut			:= T#0MS;
astBrakeReleaseTable[udiStepIndex].xEndCMD				:= FALSE;

TPL.FC_NextStep(udiStepIndex, diStep);
astBrakeReleaseTable[udiStepIndex].sTitle				:= 'Start AllSubModules';
astBrakeReleaseTable[udiStepIndex].udiModuleName		:= TPL.Gc_udiAllSubModules;
astBrakeReleaseTable[udiStepIndex].diStep				:= diStep;
astBrakeReleaseTable[udiStepIndex].diCMD				:= AXM.ET_Cmd.Start;
astBrakeReleaseTable[udiStepIndex].timTimeOut			:= T#0MS;
astBrakeReleaseTable[udiStepIndex].xEndCMD				:= FALSE;

TPL.FC_LastStep(udiStepIndex, diStep);
astBrakeReleaseTable[udiStepIndex].sTitle				:= 'End';
astBrakeReleaseTable[udiStepIndex].udiModuleName		:= 0;
astBrakeReleaseTable[udiStepIndex].diStep				:= diStep;
astBrakeReleaseTable[udiStepIndex].diCMD				:= 0;
astBrakeReleaseTable[udiStepIndex].timTimeOut			:= T#0MS;
astBrakeReleaseTable[udiStepIndex].xEndCMD				:= TRUE;

TPL.FC_NextCmdTable(iq_udiTableIndex:= udiTableIndex);
astListofCMDTables[udiTableIndex].sTitle				:= 'Brake Release';
astListofCMDTables[udiTableIndex].diCMD					:= ET_Cmd.BrakeRelease;
astListofCMDTables[udiTableIndex].udiNumberOfCmdSteps	:= udiStepIndex;

(* End of system generated code, could be modified for your application *)
END_ACTION

ACTION Init_Exceptions:
(* System generated code, could be modified for your application *)
stUpdateStructsException.etDiag												:= GD.ET_Diag.UnexpectedProgramBehavior;
stUpdateStructsException.udiDiagExt											:= ET_DiagExt.UpdateStructsException;
stUpdateStructsException.sDiagExt											:= FC_EtDiagExtToString(i_etDiagExt := stUpdateStructsException.udiDiagExt);
stUpdateStructsException.sMsg												:= '';	(* Replaced on usage *)
stUpdateStructsException.udiModuleId										:= iq_stStandardModuleItf.i_udiModuleId;
stUpdateStructsException.sModuleName										:= iq_stStandardModuleItf.i_sModuleName;
stUpdateStructsException.stReaction.axReaction[TPL.ET_Reaction.AsyncStop]	:= TRUE;
stUpdateStructsException.etSource											:= TPL.ET_ExceptionSource.NodeModule;
stUpdateStructsException.timDelayTime										:= T#0MS;
stUpdateStructsException.wHmiAttributes										:= 0;
stUpdateStructsException.xAutoQuit											:= FALSE;

stInitReactionsException.etDiag												:= GD.ET_Diag.UnexpectedProgramBehavior;
stInitReactionsException.udiDiagExt											:= ET_DiagExt.InitReactionsException;
stInitReactionsException.sDiagExt											:= FC_EtDiagExtToString(i_etDiagExt := stInitReactionsException.udiDiagExt);
stInitReactionsException.sMsg												:= '';	(* Replaced on usage *)
stInitReactionsException.udiModuleId										:= iq_stStandardModuleItf.i_udiModuleId;
stInitReactionsException.sModuleName										:= iq_stStandardModuleItf.i_sModuleName;
stInitReactionsException.stReaction.axReaction[TPL.ET_Reaction.AsyncStop]	:= TRUE;
stInitReactionsException.etSource											:= TPL.ET_ExceptionSource.NodeModule;
stInitReactionsException.timDelayTime										:= T#0MS;
stInitReactionsException.wHmiAttributes										:= 0;
stInitReactionsException.xAutoQuit											:= FALSE;

stInitSubModulesException.etDiag											:= GD.ET_Diag.UnexpectedProgramBehavior;
stInitSubModulesException.udiDiagExt										:= ET_DiagExt.InitSubModulesException;
stInitSubModulesException.sDiagExt											:= FC_EtDiagExtToString(i_etDiagExt := stInitSubModulesException.udiDiagExt);
stInitSubModulesException.sMsg												:= '';	(* Replaced on usage *)
stInitSubModulesException.udiModuleId										:= iq_stStandardModuleItf.i_udiModuleId;
stInitSubModulesException.sModuleName										:= iq_stStandardModuleItf.i_sModuleName;
stInitSubModulesException.stReaction.axReaction[TPL.ET_Reaction.AsyncStop]	:= TRUE;
stInitSubModulesException.etSource											:= TPL.ET_ExceptionSource.NodeModule;
stInitSubModulesException.timDelayTime										:= T#0MS;
stInitSubModulesException.wHmiAttributes									:= 0;
stInitSubModulesException.xAutoQuit											:= FALSE;

stIsDriveVirtualException.etDiag											:= GD.ET_Diag.InputParameterInvalid;
stIsDriveVirtualException.udiDiagExt										:= ET_DiagExt.DriveInvalid;
stIsDriveVirtualException.sDiagExt											:= FC_EtDiagExtToString(i_etDiagExt := stIsDriveVirtualException.udiDiagExt);
stIsDriveVirtualException.sMsg												:= '';	(* Replaced on usage *)
stIsDriveVirtualException.udiModuleId										:= iq_stStandardModuleItf.i_udiModuleId;
stIsDriveVirtualException.sModuleName										:= iq_stStandardModuleItf.i_sModuleName;
stIsDriveVirtualException.stReaction.axReaction[TPL.ET_Reaction.AsyncStop]	:= TRUE;
stIsDriveVirtualException.etSource											:= TPL.ET_ExceptionSource.NodeModule;
stIsDriveVirtualException.timDelayTime										:= T#0MS;
stIsDriveVirtualException.wHmiAttributes									:= 0;
stIsDriveVirtualException.xAutoQuit											:= FALSE;



(*------------------------------------------------------------------------------------------*)
(* Init User Exceptions *)

	// TPL.ET_Reaction.AsyncStop
	// TPL.ET_Reaction.SyncStopEL
	// TPL.ET_Reaction.SyncStopEH
	// TPL.ET_Reaction.StopEndOfCycle
	// TPL.ET_Reaction.MainsContactorOff

(*------------------------------------------------------------------------------------------*)
stUserException1.etDiag													:= GD.ET_Diag.ExecutionAborted;
stUserException1.udiDiagExt												:= ET_DiagExtUser.Exception1FromEquipmentModule;
stUserException1.sDiagExt												:= FC_EtDiagExtUserToString(i_etDiagExt := stUserException1.udiDiagExt);
stUserException1.sMsg													:= 'User Exception 1';
stUserException1.udiModuleId											:= iq_stStandardModuleItf.i_udiModuleId;
stUserException1.sModuleName											:= iq_stStandardModuleItf.i_sModuleName;
stUserException1.stReaction.axReaction[TPL.Gc_udiUserReactionOffset+2]	:= TRUE;
stUserException1.etSource												:= TPL.ET_ExceptionSource.User;
stUserException1.timDelayTime											:= T#0MS;
stUserException1.wHmiAttributes											:= 0;
stUserException1.xAutoQuit												:= FALSE;

stUserException2.etDiag													:= GD.ET_Diag.ExecutionAborted;
stUserException2.udiDiagExt												:= ET_DiagExtUser.Exception2FromEquipmentModule;
stUserException2.sDiagExt												:= FC_EtDiagExtUserToString(i_etDiagExt := stUserException2.udiDiagExt);
stUserException2.sMsg													:= 'User Exception 2';
stUserException2.udiModuleId											:= iq_stStandardModuleItf.i_udiModuleId;
stUserException2.sModuleName											:= iq_stStandardModuleItf.i_sModuleName;
stUserException2.stReaction.axReaction[TPL.Gc_udiUserReactionOffset+2]	:= TRUE;
stUserException2.etSource												:= TPL.ET_ExceptionSource.User;
stUserException2.timDelayTime											:= T#0MS;
stUserException2.wHmiAttributes											:= 0;
stUserException2.xAutoQuit												:= FALSE;

(* End of system generated code, could be modified for your application *)
END_ACTION

ACTION Init_Master:
(* System generated code, could be modified for your application *)

(* Standard interface *)
astSubModuleInterface[c_udiMaster].i_sModuleName	:= STANDARD.CONCAT(STR1 := iq_stStandardModuleItf.i_sModuleName, STR2 := ': Master');

astSubModuleInterface[c_udiMaster].i_xLogEnable		:= TRUE;
astSubModuleInterface[c_udiMaster].i_wLogDataFilter	:= UDINT_TO_WORD(TPL.ET_LogDataFilter.ModuleDefault);

(* AxisModule specific interface *)
stMasterInterface.stMain.i_ifMaster		:= i_ifMaster; 		(* Master *)
stMasterInterface.stMain.i_ifDrive		:= DRV_Master;
stMasterInterface.stMain.iq_lencEncoder	:= LE_Master;	


xDriveIsVirtual := FC_IsDriveVirtual(	i_ifDrive	:= stMasterInterface.stMain.i_ifDrive,
										q_etDiag	=> etDiag,
										q_etDiagExt	=> etDiagExt, //etDiagExtTPL,
										q_sMsg		=> sMsgBuffer);

IF etDiag <> GD.ET_Diag.Ok AND NOT xIsDriveVirtualException THEN										
	stIsDriveVirtualException.sMsg := sMsgBuffer;
	xIsDriveVirtualException := TRUE;
END_IF

TPL.FC_SetException(i_xExceptionActive	:= xIsDriveVirtualException, 
					iq_stException		:= stIsDriveVirtualException, 
					iq_stExceptionList	:= iq_stExceptionList, 
					iq_stLogDataList	:= iq_stLogDataList);
					
xInitSuccessful := xInitSuccessful AND NOT xIsDriveVirtualException;
etDiag := GD.ET_Diag.Ok;
	

(*Set DeadTime compensation parameters depending on used type of Master*)
FC_SetDeadTimeCompensation(i_stSubModuleInterfaceMain := stMasterInterface.stMain);
  (*Please note, FC_DeadTimeCompensation does not recognize the master type, transferred via C2C or encoder network! 
	stXXXXInterface.stMain.iq_lencEncoder.Delay must be adjusted in order to reach shaft synchronism, it depends on:
	- Transmission delay via the choosen network, depending on topology and timing 
	- Type of the master e.g. physical encoder or an axis
	- SERCOS cycle times in master and slave controllers
	
	C2C sample (similar for encoder network):
	//Access C2C_EncIn.DataDelay only if C2C_Master.SyncGroupState=5 or C2C_Slave.SyncGroupState = 5 and C2C_EncIn.DataValid = TRUE!

		//Master is a physical encoder (PMEnc/Inc):
			stXXXXInterface.stMain.iq_lencEncoder.Delay := C2C_EncIn.DataDelay - DRV_SlaveAxis.ShaftRefDelay;

		//Master is an axis (real/ virtual):
			stXXXXInterface.stMain.iq_lencEncoder.Delay := C2C_EncIn.DataDelay + one SERCOS cycle of C2C controller with connected master axis;*)


stMasterInterface.stMain.i_lrMotionActiveVelLimit						:= 15.0;		(* Limit for max. velocity of astAxisModuleInterface to switch output AxisMove in Units/s *)
stMasterInterface.stMain.i_etMotionActiveVelType						:= AXM.ET_MotionActiveVelType.Velocity;

stMasterInterface.stMain.i_timMasterStop								:= T#1S;
stMasterInterface.stMain.i_xHwLimitPos									:= FALSE;
stMasterInterface.stMain.i_xHwLimitNeg									:= FALSE;

stMasterInterface.stMain.stReducedVelocity.i_xEnableReducedVelocity		:= FALSE;
stMasterInterface.stMain.stReducedVelocity.i_xOnlyLimitCheck			:= FALSE;
stMasterInterface.stMain.stReducedVelocity.i_lrMaxReducedVelocity		:= 50.0;

stMasterInterface.stMain.i_xStart										:= FALSE;

(***************************************************************************************************************************************************************************************************)

(*** Homing ***)		
							
IF xDriveIsVirtual THEN
	stMasterInterface.stHome.i_etMode := PDL.ET_HomeMode.SetPosAxisAndLogEncoderPosition;		(* Homing Mode in case of virtual axis *)
ELSE
	stMasterInterface.stHome.i_etMode := PDL.ET_HomeMode.PosDirectionPosEdgeTp;					(* Homing Mode in case of real axis *)
END_IF


stMasterInterface.stHome.i_xEnableInitAbsReadPos := TRUE;						(* TRUE : Restores the AxisPosition depending on the stHome.etMode
																						  If stHome.i_etMode is equal to PDL.ET_HomeMode.RestorePosFromAxisEncoder or 
																						  to PDL.ET_HomeMode.WriteAxisEncoder, the encoder of the axis is read,
																						  or else the position will be restored from the retain area *)

stMasterInterface.stHome.stSetpos.iq_pstRestorePosRetain := ADR(Grp_stRestorePositionAxis1);

stMasterInterface.stHome.i_xResetHomeOk := FALSE;

(* Possible modes for homing mode Sensor:
	PDL.ET_HomeMode.PosDirectionPosEdgeSensor
	PDL.ET_HomeMode.NegDirectionPosEdgeSensor
	PDL.ET_HomeMode.NegDirectionNegEdgeSensor
	PDL.ET_HomeMode.PosDirectionNegEdgeSensor
*)
stMasterInterface.stHome.stSensor.i_lrHomePosition			:= 0.0;			(* Position at the end of homing in units *)
stMasterInterface.stHome.stSensor.i_lrVel					:= 10.0;		(* Homing ceiling velocity in units/s *)
stMasterInterface.stHome.stSensor.i_lrAcc					:= 1000.0;		(* Homing acceleration in units/s^2 *)
stMasterInterface.stHome.stSensor.i_lrDec					:= 1000.0;		(* Homing deceleration in units/s^2 *)
stMasterInterface.stHome.stSensor.i_lrJerk					:= 10000.0;		(* Homing jerk in units/s^3 *)
stMasterInterface.stHome.stSensor.i_lrOffset				:= 0.0;			(* Offset from home signal in units *)
stMasterInterface.stHome.stSensor.i_lrMaxTravel 			:= 720.0;		(* Max. travel for referencing by normal input *)
stMasterInterface.stHome.stSensor.i_xRotativeSystem			:= FALSE;		(* Rotative system true or false for referencing by normal input *)
stMasterInterface.stHome.stSensor.i_xSensor 				:= FALSE;		(* Input for home signal. Can be a signal from a controller input. Has to be written cyclic. *)

(* Possible Modes for homing mode LimitSwitch:
	PDL.ET_HomeMode.PosDirectionPosEdgeHWLimitPos		normally open contact / Closing contact
	PDL.ET_HomeMode.NegDirectionPosEdgeHWLimitNeg		normally open contact / Closing contact
	PDL.ET_HomeMode.NegDirectionNegEdgeHWLimitNeg		normally closed contact / Opening contact  
	PDL.ET_HomeMode.PosDirectionNegEdgeHWLimitPos		normally closed contact / Opening contact 
*)
stMasterInterface.stHome.stLimitSwitch.i_lrHomePosition 	:= 0.0;			(* Position at the end of homing in units *)
stMasterInterface.stHome.stLimitSwitch.i_lrVel				:= 10.0;		(* Homing ceiling velocity in units/s *)
stMasterInterface.stHome.stLimitSwitch.i_lrLowVel			:= 5.0;			(* Homing low ceiling velocity in units/s *)
stMasterInterface.stHome.stLimitSwitch.i_lrAcc				:= 1000.0;		(* Homing acceleration in units/s^2 *)
stMasterInterface.stHome.stLimitSwitch.i_lrDec				:= 1000.0;		(* Homing deceleration in units/s^2 *)
stMasterInterface.stHome.stLimitSwitch.i_lrJerk				:= 10000.0;		(* Homing jerk in units/s^3 *)
stMasterInterface.stHome.stLimitSwitch.i_lrOffset			:= 0.0;			(* Offset from home signal in units *)
stMasterInterface.stHome.stLimitSwitch.i_lrMaxTravel 		:= 9999.0;		(* Max. travel for referencing normal input as a hardware limit *)

(* Possible modes for homing mode MoveOnPos:
	PDL.ET_HomeMode.MoveOnPosAbs 
*)
stMasterInterface.stHome.stMoveOnPos.i_lrTarget				:= 0.0;			(* Position at the end of homing in units *)
stMasterInterface.stHome.stMoveOnPos.i_lrVel				:= 10.0;		(* Homing ceiling velocity in units/s *)
stMasterInterface.stHome.stMoveOnPos.i_lrAcc				:= 1000.0;		(* Homing acceleration in units/s^2 *)
stMasterInterface.stHome.stMoveOnPos.i_lrDec				:= 1000.0;		(* Homing deceleration in units/s^2 *)
stMasterInterface.stHome.stMoveOnPos.i_lrJerk				:= 10000.0;		(* Homing jerk in units/s^3 *)
stMasterInterface.stHome.stMoveOnPos.i_lrPeriod				:= 0.0;			(* Period of the axis *)
stMasterInterface.stHome.stMoveOnPos.i_xRotativeSystem		:= FALSE;		(* Rotative system true or false *)

(* Possible modes for homing mode SetPos:
	PDL.ET_HomeMode.SetPosAxisPosition 
	PDL.ET_HomeMode.SetPosLogEncoderPosition 
	PDL.ET_HomeMode.SetPosAxisAndLogEncoderPosition
	PDL.ET_HomeMode.RestorePosFromAxisEncoder 
	PDL.ET_HomeMode.RestorePosFromRetain 
*)
stMasterInterface.stHome.stSetpos.i_lrHomePosition			:= 0.0;			(* Position at the end of homing in units *)
stMasterInterface.stHome.stSetpos.i_lrEncoderPosition		:= 0.0;			(* Encoder position in units after homing *)
stMasterInterface.stHome.stSetpos.i_lrAbsEncOffset			:= 100.0;		(* Distance to the jump of axis encoder in units *)
stMasterInterface.stHome.stSetpos.i_lrRestoreWindow			:= 180;			(* How far can the drive be away from its correct position *)
stMasterInterface.stHome.stSetpos.i_lrUserPeriod			:= 360;			(* Period of the axis *)

(* Possible modes for homing mode Torque:
	PDL.ET_HomeMode.PosDirectionMaxTorque 
	PDL.ET_HomeMode.NegDirectionMaxTorque 
*)
stMasterInterface.stHome.stTorque.i_lrHomePosition			:= 0.0;			(* Position at the end of homing in units *)
stMasterInterface.stHome.stTorque.i_lrVel					:= 10.0;		(* Homing ceiling velocity in units/s *)
stMasterInterface.stHome.stTorque.i_lrAcc					:= 1000.0;		(* Homing acceleration in units/s^2 *)
stMasterInterface.stHome.stTorque.i_lrDec					:= 1000.0;		(* Homing deceleration in units/s^2 *)
stMasterInterface.stHome.stTorque.i_lrJerk					:= 10000.0;		(* Homing jerk in units/s^3 *)
stMasterInterface.stHome.stTorque.i_lrOffset				:= 0.0;			(* Offset from home signal in units *)
stMasterInterface.stHome.stTorque.i_lrMaxTravel				:= 9999.0;		(* Max. travel for referencing by torque *)
stMasterInterface.stHome.stTorque.i_lrMaxTorque				:= 0.0;			(* Torque for stop in Nm / referencing by torque *)
stMasterInterface.stHome.stTorque.i_diTorqueTime			:= 5;			(* Time in msec to hold torque *)

(* Possible modes for homing mode TouchProbe:
	PDL.ET_HomeMode.PosDirectionPosEdgeTp 
	PDL.ET_HomeMode.NegDirectionPosEdgeTp 
	PDL.ET_HomeMode.NegDirectionNegEdgeTp 
	PDL.ET_HomeMode.PosDirectionNegEdgeTp 
*)
stMasterInterface.stHome.stTouchProbe.i_lrHomePosition		:= 0.0;			(* Position at the end of homing in units *)
stMasterInterface.stHome.stTouchProbe.i_lrVel				:= 100.0;		(* Homing ceiling velocity in units/s *)
stMasterInterface.stHome.stTouchProbe.i_lrAcc				:= 1000.0;		(* Homing acceleration in units/s^2 *)
stMasterInterface.stHome.stTouchProbe.i_lrDec				:= 1000.0;		(* Homing deceleration in units/s^2 *)
stMasterInterface.stHome.stTouchProbe.i_lrJerk				:= 10000.0;		(* Homing jerk in units/s^3 *)
stMasterInterface.stHome.stTouchProbe.i_lrOffset			:= 30.0;		(* Offset from home signal in units *)
stMasterInterface.stHome.stTouchProbe.i_lrMaxTravel			:= 720.0;		(* Max. travel for referencing by TP *)
stMasterInterface.stHome.stTouchProbe.i_xRotativeSystem		:= TRUE;		(* Rotative system true or false for referencing by TP *)
stMasterInterface.stHome.stTouchProbe.i_ifTouchProbe		:= TP_0;		(* Input for TP *)

(* Possible modes for homing mode WritePos:
	PDL.ET_HomeMode.WriteAxisEncoder 
*)
stMasterInterface.stHome.stWritePos.i_lrHomePosition		:= 0.0;			(* Position at the end of homing in units *)
stMasterInterface.stHome.stWritePos.i_lrUserPeriod			:= 0.0;			(* Calculates Drive.Position into period ( units ) *)
stMasterInterface.stHome.stWritePos.i_lrAbsEncOffset		:= 100.0;		(* Distance to the jump of axis encoder in units *)

(***************************************************************************************************************************************************************************************************)
(*** Manual ***)

stMasterInterface.stManual.i_lrVel								:= 50.0;			(* Velocity in units/s *)
stMasterInterface.stManual.i_lrAcc								:= 100.0;			(* Acceleration in units/s^2 *)
stMasterInterface.stManual.i_lrDec								:= 100.0;			(* Deceleration in units/s^2 *)
stMasterInterface.stManual.i_lrJerk								:= 1000.0;			(* Jerk in units/s^3 *)
stMasterInterface.stManual.i_lrMaxDistance						:= 120.0;			(* Max pathlengths for one step in units *)
stMasterInterface.stManual.i_xEndless							:= FALSE;			(* TRUE: jogging endless; Position between the periode; FALSE: jogging in steps. Position can be out of periode *)
stMasterInterface.stManual.i_lrPeriod							:= 360.0;			(* Period of the axis *)

(***************************************************************************************************************************************************************************************************)
(*** Cam ***)

stMasterInterface.stMultiCam.i_etCSModeSlave					:= PDL.ET_MultiCamCsModeSlave.SetSlavePositionToFirstCamPosition;		(* ColdStartMode Slave *)
stMasterInterface.stMultiCam.i_etCSModeMaster					:= PDL.ET_MultiCamCsModeMaster.SetMasterPositionToFirstCamPosition;		(* ColdStartMode Master *)
stMasterInterface.stMultiCam.i_etWSMode							:= PDL.ET_MultiCamWsMode.StoredCamMoveAlwaysNoPositionCheck;			(* WarmStartMode *)
stMasterInterface.stMultiCam.i_lrWSWindow						:= 5.0;											(* WarmStartWindow in Axis units *)
stMasterInterface.stMultiCam.i_lrWSVel							:= 10.0;										(* Velocity for WarmStart and CSModeSlave = PDL.ET_MultiCamCsModeSlave.MoveSlaveToFirstCamPosition in Units/s *)
stMasterInterface.stMultiCam.i_lrWSAcc							:= 1000.0;										(* Acceleration and deceleration for Warmstart and CSModeSlave = PDL.ET_MultiCamCsModeSlave.MoveSlaveToFirstCamPosition in Units/s^2 *)
stMasterInterface.stMultiCam.i_lrWSJerk							:= 10000.0;										(* Jerk for Warmstart and CSModeSlave = PDL.ET_MultiCamCsModeSlave.MoveSlaveToFirstCamPosition in units/s^3 *)
stMasterInterface.stMultiCam.i_diTXend							:= 2*SYSTEMINTERFACE.FC_LzsTaskGetInterval();	(* Time of XLowEnd and XHighEnd befor Xend or Xstart in msec*)
stMasterInterface.stMultiCam.i_lrInstantXLimMax					:= 0.0;											(* Switch off position at 'InstantNewCam' *)

stMasterInterface.stMultiCam.i_xEnableTabHandler				:= TRUE;										(* TRUE: TabHandler is enabled *)
stMasterInterface.stMultiCam.i_udiTableSelectNr					:= AXM.ET_ParId.User;							(* Number of table which is used in the next cycle *)								

stMasterInterface.stMultiCam.i_xSetEncoderParameters			:= FALSE;										(* TRUE: The parameters MasterId, FeedConstand, GearIn and GearOut will be copyed into LEnc object *)
stMasterInterface.stMultiCam.i_xSetEncoderPosition				:= FALSE;										(* TRUE: Manipulation of LEnc object on startup OpMode MultiCam *)
stMasterInterface.stMultiCam.i_lrSetEncoderOffset				:= 0.0;											(* Master encoder offset *)
stMasterInterface.stMultiCam.i_xCheckEncoderPeriod				:= TRUE;										(* TRUE: Check of encoder period = 0. If encoder period <> 0 -> Exception *)

stMasterInterface.stMultiCam.iq_astMotionPar[AXM.ET_ParId.User].diNumberOfCamPoints			:= 4;	(* DataStruct for the next cycle *)
stMasterInterface.stMultiCam.iq_astMotionPar[AXM.ET_ParId.User].lrYPeriod					:= 0.0;

stMasterInterface.stMultiCam.iq_astMotionPar[AXM.ET_ParId.User].astCamPoint[0].lrX			:= 0.0;
stMasterInterface.stMultiCam.iq_astMotionPar[AXM.ET_ParId.User].astCamPoint[0].lrY			:= 0.0;
stMasterInterface.stMultiCam.iq_astMotionPar[AXM.ET_ParId.User].astCamPoint[0].lrM			:= 0.0;
stMasterInterface.stMultiCam.iq_astMotionPar[AXM.ET_ParId.User].astCamPoint[0].etCamType	:= PDL.ET_CamType.Poly5Com;
stMasterInterface.stMultiCam.iq_astMotionPar[AXM.ET_ParId.User].astCamPoint[1].lrX			:= 60.0;
stMasterInterface.stMultiCam.iq_astMotionPar[AXM.ET_ParId.User].astCamPoint[1].lrY			:= 30.0;
stMasterInterface.stMultiCam.iq_astMotionPar[AXM.ET_ParId.User].astCamPoint[1].lrM			:= 1.0;
stMasterInterface.stMultiCam.iq_astMotionPar[AXM.ET_ParId.User].astCamPoint[1].etCamType	:= PDL.ET_CamType.Straight;
stMasterInterface.stMultiCam.iq_astMotionPar[AXM.ET_ParId.User].astCamPoint[2].lrX			:= 240.0;
stMasterInterface.stMultiCam.iq_astMotionPar[AXM.ET_ParId.User].astCamPoint[2].lrY			:= 210.0;
stMasterInterface.stMultiCam.iq_astMotionPar[AXM.ET_ParId.User].astCamPoint[2].lrM			:= 1.0;
stMasterInterface.stMultiCam.iq_astMotionPar[AXM.ET_ParId.User].astCamPoint[2].etCamType	:= PDL.ET_CamType.Poly5Com;
stMasterInterface.stMultiCam.iq_astMotionPar[AXM.ET_ParId.User].astCamPoint[3].lrX			:= 360.0;
stMasterInterface.stMultiCam.iq_astMotionPar[AXM.ET_ParId.User].astCamPoint[3].lrY			:= 0.0;
stMasterInterface.stMultiCam.iq_astMotionPar[AXM.ET_ParId.User].astCamPoint[3].lrM			:= 0.0;
stMasterInterface.stMultiCam.iq_astMotionPar[AXM.ET_ParId.User].astCamPoint[3].etCamType	:= PDL.ET_CamType.Poly5Com;

stMasterInterface.stMultiCam.iq_astMotionPar[AXM.ET_ParId.Idle].diUserTableId	:= UDINT_TO_DINT(AXM.ET_ParId.Idle);
stMasterInterface.stMultiCam.iq_astMotionPar[AXM.ET_ParId.Start].diUserTableId	:= UDINT_TO_DINT(AXM.ET_ParId.Start);
stMasterInterface.stMultiCam.iq_astMotionPar[AXM.ET_ParId.Cont].diUserTableId	:= UDINT_TO_DINT(AXM.ET_ParId.Cont);
stMasterInterface.stMultiCam.iq_astMotionPar[AXM.ET_ParId.Stop].diUserTableId	:= UDINT_TO_DINT(AXM.ET_ParId.Stop);
stMasterInterface.stMultiCam.iq_astMotionPar[AXM.ET_ParId.User].diUserTableId	:= UDINT_TO_DINT(AXM.ET_ParId.User);


(***************************************************************************************************************************************************************************************************)
(*** Endless ***)

stMasterInterface.stEndless.i_lrVel								:= 100.0;			(* Velocity in Units/s *)
stMasterInterface.stEndless.i_lrAcc								:= 1000.0;			(* Acceleration in Units/s^2 *)
stMasterInterface.stEndless.i_lrDec								:= 1000.0;			(* Deceleration in Units/s^2 *)
stMasterInterface.stEndless.i_lrJerk							:= 10000.0;			(* Jerk in units/s^3 *)
stMasterInterface.stEndless.i_lrPeriod							:= 360.0;			(* Period one cycle in units *)
stMasterInterface.stEndless.i_lrStopPosition					:= 0.5;				(* Stop position in units *)


(***************************************************************************************************************************************************************************************************)
(*** Pos ***)

stMasterInterface.stPos.i_etPosMode								:= SYSTEMINTERFACE.ET_PosMode.Endless;		(* SYSTEMINTERFACE.ET_PosMode.Endless, SYSTEMINTERFACE.ET_PosMode.Relative, SYSTEMINTERFACE.ET_PosMode.Absolute *)
stMasterInterface.stPos.i_lrTarget								:= 360.0;									(* Target position or distance in Units *)
stMasterInterface.stPos.i_lrVel									:= 360.0;									(* Ceiling velocity in Units/s *)
stMasterInterface.stPos.i_lrAcc									:= 3600.0;									(* Acceleration in Units/s^2 *)
stMasterInterface.stPos.i_lrDec									:= 3600.0;									(* Deceleration in Units/s^2 *)
stMasterInterface.stPos.i_lrJerk								:= 36000.0;									(* Jerk in units/s^3 *)

(* End of system generated code, could be modified for your application *)
END_ACTION

ACTION Init_Reactions:
(* System generated code, only to be changed by experienced programmers *)
IF c_udiNumberOfSubModules < 1 THEN
	RETURN;
END_IF

(* Change of default reactions only on demand *)
(* Compare SR MainMachine Action Init_Reactions *)

xInitReactionsException := FALSE;

(*****************************************************************************************************************************************************)
(* Init ReactionTranslationMode *)

TPL.FC_InitReactionTranslationMode(	i_udiNumberOfSubModules			:= c_udiNumberOfSubModules,
									i_petReactionTranslationMode	:= ADR(aetReactionTranslationMode),
									q_etDiag						=> etDiag,
									q_etDiagExt						=> etDiagExtTPL);
							
IF etDiag <> GD.ET_Diag.Ok AND NOT xInitReactionsException THEN
	xInitReactionsException := TRUE;
	
	stInitReactionsException.sMsg := PDL.FC_MultiConcat(i_sString1 := 'InitReactionTranslationMode - ', 
														i_sString2 := GD.FC_EtDiagToString(i_etDiag := etDiag), 
														i_sString3 := ' - ', 
														i_sString4 := TPL.FC_EtDiagExtToString(i_etDiagExt := etDiagExtTPL));
END_IF	

(*****************************************************************************************************************************************************)
(* Init ReactionTranslationTable *)	

TPL.FC_InitReactionTranslationTable(i_udiNumberOfSubModules			:= c_udiNumberOfSubModules,
									i_pstReactionTranslationTable	:= ADR(aastReactionTranslationTable),
									q_etDiag						=> etDiag,
									q_etDiagExt						=> etDiagExtTPL);
									
IF etDiag <> GD.ET_Diag.Ok AND NOT xInitReactionsException THEN
	xInitReactionsException := TRUE;
	
	stInitReactionsException.sMsg := PDL.FC_MultiConcat(i_sString1 := 'InitReactionTranslationTable - ', 
														i_sString2 := GD.FC_EtDiagToString(i_etDiag := etDiag), 
														i_sString3 := ' - ', 
														i_sString4 := TPL.FC_EtDiagExtToString(i_etDiagExt := etDiagExtTPL));
END_IF		

(*****************************************************************************************************************************************************)
(* Init ReactionTranslationJobs *)	
					
TPL.FC_InitReactionTranslationJobs( i_udiNumberOfSubModules			:= c_udiNumberOfSubModules,
									i_pstReactionTranslationJobs	:= ADR(astReactionTranslationJobs),
									q_etDiag						=> etDiag,
									q_etDiagExt						=> etDiagExtTPL);
						
IF etDiag <> GD.ET_Diag.Ok AND NOT xInitReactionsException THEN
	xInitReactionsException := TRUE;
	
	stInitReactionsException.sMsg := PDL.FC_MultiConcat(i_sString1 := 'InitReactionTranslationJobs - ', 
														i_sString2 := GD.FC_EtDiagToString(i_etDiag := etDiag), 
														i_sString3 := ' - ', 
														i_sString4 := TPL.FC_EtDiagExtToString(i_etDiagExt := etDiagExtTPL));
END_IF		

(*****************************************************************************************************************************************************)
(* Set exception if any exception occurred *)

TPL.FC_SetException(i_xExceptionActive	:= xInitReactionsException, 
					iq_stException		:= stInitReactionsException, 
					iq_stExceptionList	:= iq_stExceptionList, 
					iq_stLogDataList	:= iq_stLogDataList);
					
xInitSuccessful := xInitSuccessful AND NOT xInitReactionsException;

etDiag := GD.ET_Diag.Ok;
(* End of system generated code, only to be changed by experienced programmers *)
END_ACTION

ACTION Init_SubModules:
(* System generated code, could be modified for your application *)

(* Module Group declaration *)

(* aaudiSubModuleGroups[c_udiAlphaGroup1-TPL.Gc_udiGroupOffset,TPL.ET_Group.Member1]	:= c_udiMaster; *)	(* The c_diMaster is the first element of the group c_diAlphaGroup1 *)
(* aaudiSubModuleGroups[c_udiAlphaGroup1-TPL.Gc_udiGroupOffset,TPL.ET_Group.Member2]	:= 0;			*)	(* There is no second element of the group c_diAlphaGroup1 *)

(* aaudiSubModuleGroups[c_udiAlphaGroup2-TPL.Gc_udiGroupOffset,TPL.ET_Group.Member1]	:= 0;			*)	(* There is no first element of the group c_diAlphaGroup2 *)
(* aaudiSubModuleGroups[c_udiAlphaGroup2-TPL.Gc_udiGroupOffset,TPL.ET_Group.Member2]	:= 0;			*)	(* There is no second element of the group c_diAlphaGroup2 *)

(* End of system generated code, could be modified for your application *)


(* System generated code, do not change without consulting 'Schneider Electric Automation GmbH' - otherwise you risk instability!!!*)
xInitSubModulesException := FALSE;

(*****************************************************************************************************************************************************)
(* Set IDs of SubModules *)	

TPL.FC_SetSubModuleIds(	i_udiMainModuleId			:= iq_stStandardModuleItf.i_udiModuleId,
						i_pstSubModulesItf			:= ADR(astSubModuleInterface),
						i_udiNumberOfSubModules		:= c_udiNumberOfSubModules,
						q_etDiag					=> etDiag,
						q_etDiagExt					=> etDiagExtTPL);
					
IF etDiag <> GD.ET_Diag.Ok AND NOT xInitSubModulesException THEN
	xInitSubModulesException := TRUE;
	
	stInitSubModulesException.sMsg := PDL.FC_MultiConcat(	i_sString1 := 'SetSubModuleIds - ', 
															i_sString2 := GD.FC_EtDiagToString(i_etDiag := etDiag), 
															i_sString3 := ' - ', 
															i_sString4 := TPL.FC_EtDiagExtToString(i_etDiagExt := etDiagExtTPL));
END_IF	

(*****************************************************************************************************************************************************)
(* Set exception if any exception occurred *)

TPL.FC_SetException(i_xExceptionActive	:= xInitSubModulesException, 
					iq_stException		:= stInitSubModulesException, 
					iq_stExceptionList	:= iq_stExceptionList, 
					iq_stLogDataList	:= iq_stLogDataList);

xInitSuccessful := xInitSuccessful AND NOT xInitSubModulesException;
					
etDiag := GD.ET_Diag.Ok;
(* End of system generated code, do not change without consulting 'Schneider Electric Automation GmbH' - otherwise you risk instability!!!*)
END_ACTION

ACTION InitModule_Action:
(* This step is used for initialisations after being enabled *)

(* System generated code, could be modified for your application *)
Init_Exceptions();
(* End of system generated code, could be modified for your application *)

(* System generated code, do not change without consulting 'Schneider Electric Automation GmbH' - otherwise you risk instability!!!*)
xInitSuccessful := TRUE;
xIsDriveVirtualException := FALSE;

iq_stStandardModuleItf.q_xActive		:= TRUE;
iq_stStandardModuleItf.q_xReady			:= FALSE;
iq_stStandardModuleItf.q_etDiag			:= GD.ET_Diag.Ok;
iq_stStandardModuleItf.q_udiDiagExt		:= ET_DiagExt.Initializing;
iq_stStandardModuleItf.q_sDiagExt		:= FC_EtDiagExtToString(i_etDiagExt := ET_DiagExt.Initializing);
iq_stStandardModuleItf.q_sMsg			:= '';
			
Init_SubModules();
Init_CmdTables();
Init_Reactions();
UpdateStructs();
(* End of system generated code, do not change without consulting 'Schneider Electric Automation GmbH' - otherwise you risk instability!!!*)

(* System generated code, could be modified for your application *)
Init_Master();
(* End of system generated code, could be modified for your application *)

(* Application specific code *)
(* ToDo: Add your application specific code here *)
;
(* End of application specific code *)
END_ACTION

ACTION Input_Action:
(* System generated code, do not change without consulting 'Schneider Electric Automation GmbH' - otherwise you risk instability!!!*)
UpdateStructs();
(* End of system generated code, do not change without consulting 'Schneider Electric Automation GmbH' - otherwise you risk instability!!!*)
END_ACTION

ACTION Logger_Action:
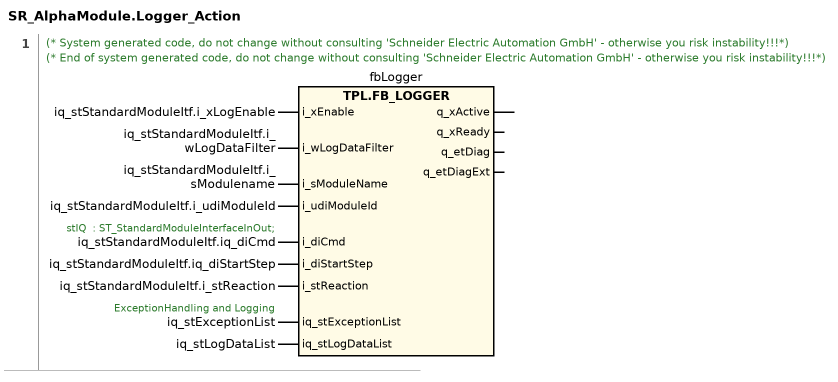
// NETWORK 1
// 					(* System generated code, do not change without consulting 'Schneider Electric Automation GmbH' - otherwise you risk instability!!!*)
// (* End of system generated code, do not change without consulting 'Schneider Electric Automation GmbH' - otherwise you risk instability!!!*)
//
//   fbLogger: Logging related variables
//   iq_stStandardModuleItf.iq_diCmd: stIQ : ST_StandardModuleInterfaceInOut;
//   iq_stExceptionList: ExceptionHandling and Logging
fbLogger(
    i_xEnable := iq_stStandardModuleItf.i_xLogEnable,
    i_wLogDataFilter := iq_stStandardModuleItf.i_wLogDataFilter,
    i_sModuleName := iq_stStandardModuleItf.i_sModulename,
    i_udiModuleId := iq_stStandardModuleItf.i_udiModuleId,
    i_diCmd := iq_stStandardModuleItf.iq_diCmd,
    i_diStartStep := iq_stStandardModuleItf.iq_diStartStep,
    i_stReaction := iq_stStandardModuleItf.i_stReaction,
    iq_stExceptionList := iq_stExceptionList,
    iq_stLogDataList := iq_stLogDataList); // TPL.FB_LOGGER
END_ACTION

ACTION ModuleFaults:
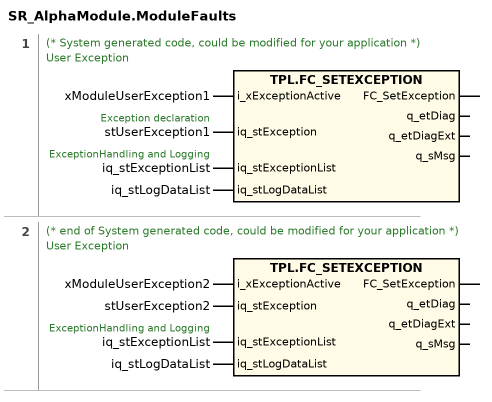
// NETWORK 1
// (* System generated code, could be modified for your application *)
// User Exception
//   stUserException1: Exception declaration
//   iq_stExceptionList: ExceptionHandling and Logging
TPL.FC_SETEXCEPTION(i_xExceptionActive := xModuleUserException1, iq_stException := stUserException1, iq_stExceptionList := iq_stExceptionList, iq_stLogDataList := iq_stLogDataList);

// NETWORK 2
// (* end of System generated code, could be modified for your application *)
// User Exception
//   iq_stExceptionList: ExceptionHandling and Logging
TPL.FC_SETEXCEPTION(i_xExceptionActive := xModuleUserException2, iq_stException := stUserException2, iq_stExceptionList := iq_stExceptionList, iq_stLogDataList := iq_stLogDataList);
END_ACTION

ACTION Output_Active:
(* System generated code, only to be changed by experienced programmers *)
IF iq_stStandardModuleItf.q_udiSubModuleInException <> 0 THEN
	iq_stStandardModuleItf.q_etDiag		:= GD.ET_Diag.Ok;
	iq_stStandardModuleItf.q_udiDiagExt	:= ET_DiagExt.SubModuleInException;
	iq_stStandardModuleItf.q_sDiagExt		:= FC_EtDiagExtToString(i_etDiagExt := ET_DiagExt.SubModuleInException);
	iq_stStandardModuleItf.q_sMsg			:= '';
ELSE
	IF etDiagModuleController = GD.ET_Diag.Ok THEN
		iq_stStandardModuleItf.q_etDiag	:= etDiagModuleController;
		iq_stStandardModuleItf.q_sMsg		:= sMsgModuleController;
		
		CASE etDiagExtModuleController OF
			TPL.ET_DiagExt.DeactivatingSubModules : 
				iq_stStandardModuleItf.q_udiDiagExt	:= ET_DiagExt.DeactivatingSubModules;
				iq_stStandardModuleItf.q_sDiagExt		:= FC_EtDiagExtToString(i_etDiagExt := ET_DiagExt.DeactivatingSubModules);
			TPL.ET_DiagExt.Disabled : 
				iq_stStandardModuleItf.q_udiDiagExt	:= ET_DiagExt.Disabled;
				iq_stStandardModuleItf.q_sDiagExt		:= FC_EtDiagExtToString(i_etDiagExt := ET_DiagExt.Disabled);
			TPL.ET_DiagExt.ExecuteStep : 
				iq_stStandardModuleItf.q_udiDiagExt	:= ET_DiagExt.ExecuteStep;
				iq_stStandardModuleItf.q_sDiagExt		:= FC_EtDiagExtToString(i_etDiagExt := ET_DiagExt.ExecuteStep);
			TPL.ET_DiagExt.Initializing : 
				iq_stStandardModuleItf.q_udiDiagExt	:= ET_DiagExt.Initializing;
				iq_stStandardModuleItf.q_sDiagExt		:= FC_EtDiagExtToString(i_etDiagExt := ET_DiagExt.Initializing);
			TPL.ET_DiagExt.WaitAtNegativeStep : 
				iq_stStandardModuleItf.q_udiDiagExt	:= ET_DiagExt.WaitAtNegativeStep;
				iq_stStandardModuleItf.q_sDiagExt		:= FC_EtDiagExtToString(i_etDiagExt := ET_DiagExt.WaitAtNegativeStep);
			TPL.ET_DiagExt.WaitCmdsDone : 
				iq_stStandardModuleItf.q_udiDiagExt	:= ET_DiagExt.WaitCmdsDone;
				iq_stStandardModuleItf.q_sDiagExt		:= FC_EtDiagExtToString(i_etDiagExt := ET_DiagExt.WaitCmdsDone);
			TPL.ET_DiagExt.WaitForCmd : 
				iq_stStandardModuleItf.q_udiDiagExt	:= ET_DiagExt.WaitForCmd;
				iq_stStandardModuleItf.q_sDiagExt		:= FC_EtDiagExtToString(i_etDiagExt := ET_DiagExt.WaitForCmd);
			ELSE
				iq_stStandardModuleItf.q_etDiag		:= GD. ET_Diag.UnexpectedProgramBehavior;
				iq_stStandardModuleItf.q_udiDiagExt	:= ET_DiagExt.UnknownStateModuleController;
				iq_stStandardModuleItf.q_sDiagExt		:= FC_EtDiagExtToString(i_etDiagExt := ET_DiagExt.UnknownStateModuleController);
		END_CASE
	ELSE
		iq_stStandardModuleItf.q_etDiag		:= GD.ET_Diag.DiagActive;
		iq_stStandardModuleItf.q_udiDiagExt	:= ET_DiagExt.ModuleControllerException;
		iq_stStandardModuleItf.q_sDiagExt		:= FC_EtDiagExtToString(i_etDiagExt := ET_DiagExt.ModuleControllerException);
		iq_stStandardModuleItf.q_sMsg			:= PDL.FC_MultiConcat(	i_sString1 := GD.FC_EtDiagToString(i_etDiag := etDiagModuleController), 
																			i_sString2 := ' - ',
																			i_sString3 := TPL.FC_EtDiagExtToString(i_etDiagExt := etDiagExtModuleController), 
																			i_sString4 := '');
	END_IF
END_IF

(* End of system generated code, only to be changed by experienced programmers *)
END_ACTION

ACTION Start_Action:
(* This step is active until the machine is being enabled *)

(* System generated code, do not change without consulting 'Schneider Electric Automation GmbH' - otherwise you risk instability!!! *)
iq_stStandardModuleItf.q_xActive			:= FALSE;
iq_stStandardModuleItf.q_xReady				:= FALSE;

iq_stStandardModuleItf.q_etDiag				:= GD.ET_Diag.Ok;
iq_stStandardModuleItf.q_udiDiagExt			:= ET_DiagExt.Disabled;
iq_stStandardModuleItf.q_sDiagExt			:= FC_EtDiagExtToString(i_etDiagExt := iq_stStandardModuleItf.q_udiDiagExt);
iq_stStandardModuleItf.q_sMsg				:= '';

iq_stStandardModuleItf.q_dwModuleType		:= TPL.ET_ModuleType.NodeModule;
iq_stStandardModuleItf.q_sModuleTypeName	:= 'NodeModule';
iq_stStandardModuleItf.q_udiModuleVersion	:= 1;	
(* End of system generated code, do not change without consulting 'Schneider Electric Automation GmbH' - otherwise you risk instability!!! *)

(* System generated code, to be changed by experienced programmers *)
IF iq_stStandardModuleItf.iq_diCmd <> 0 AND NOT iq_stStandardModuleItf.i_xEnable THEN
	iq_stStandardModuleItf.iq_diCmd := 0;
END_IF
(* End of system generated code, to be changed by experienced programmers *)

(* Application specific code *)
(* ToDo: Add your application specific code here *)
;
(* End of application specific code *)
END_ACTION

ACTION SubModules_Action:
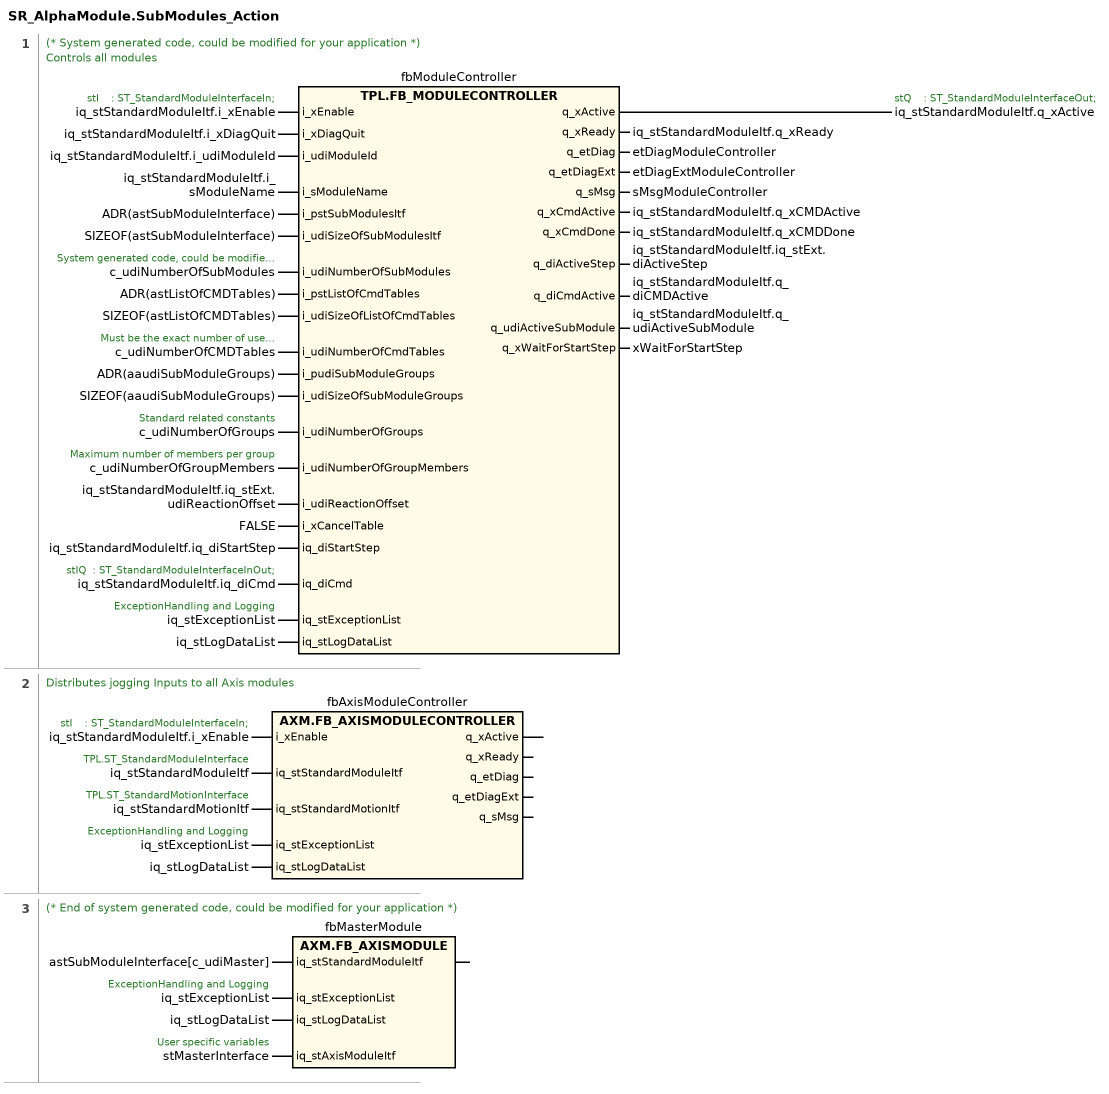
// NETWORK 1
// 					(* System generated code, could be modified for your application *)
// Controls all modules
//
//   fbModuleController: Modules related variables
//   iq_stStandardModuleItf.i_xEnable: stI : ST_StandardModuleInterfaceIn;
//   c_udiNumberOfSubModules: System generated code, could be modified for your application
//   c_udiNumberOfCMDTables: Must be the exact number of used CmdTables!
//   c_udiNumberOfGroups: Standard related constants
//   c_udiNumberOfGroupMembers: Maximum number of members per group
//   iq_stStandardModuleItf.iq_diCmd: stIQ : ST_StandardModuleInterfaceInOut;
//   iq_stExceptionList: ExceptionHandling and Logging
//   iq_stStandardModuleItf.q_xActive: stQ : ST_StandardModuleInterfaceOut;
fbModuleController(
    i_xEnable := iq_stStandardModuleItf.i_xEnable,
    i_xDiagQuit := iq_stStandardModuleItf.i_xDiagQuit,
    i_udiModuleId := iq_stStandardModuleItf.i_udiModuleId,
    i_sModuleName := iq_stStandardModuleItf.i_sModuleName,
    i_pstSubModulesItf := ADR(astSubModuleInterface),
    i_udiSizeOfSubModulesItf := SIZEOF(astSubModuleInterface),
    i_udiNumberOfSubModules := c_udiNumberOfSubModules,
    i_pstListOfCmdTables := ADR(astListOfCMDTables),
    i_udiSizeOfListOfCmdTables := SIZEOF(astListOfCMDTables),
    i_udiNumberOfCmdTables := c_udiNumberOfCMDTables,
    i_pudiSubModuleGroups := ADR(aaudiSubModuleGroups),
    i_udiSizeOfSubModuleGroups := SIZEOF(aaudiSubModuleGroups),
    i_udiNumberOfGroups := c_udiNumberOfGroups,
    i_udiNumberOfGroupMembers := c_udiNumberOfGroupMembers,
    i_udiReactionOffset := iq_stStandardModuleItf.iq_stExt.udiReactionOffset,
    i_xCancelTable := FALSE,
    iq_diStartStep := iq_stStandardModuleItf.iq_diStartStep,
    iq_diCmd := iq_stStandardModuleItf.iq_diCmd,
    iq_stExceptionList := iq_stExceptionList,
    iq_stLogDataList := iq_stLogDataList,
    q_xReady => iq_stStandardModuleItf.q_xReady,
    q_etDiag => etDiagModuleController,
    q_etDiagExt => etDiagExtModuleController,
    q_sMsg => sMsgModuleController,
    q_xCmdActive => iq_stStandardModuleItf.q_xCMDActive,
    q_xCmdDone => iq_stStandardModuleItf.q_xCMDDone,
    q_diActiveStep => iq_stStandardModuleItf.iq_stExt.diActiveStep,
    q_diCmdActive => iq_stStandardModuleItf.q_diCMDActive,
    q_udiActiveSubModule => iq_stStandardModuleItf.q_udiActiveSubModule,
    q_xWaitForStartStep => xWaitForStartStep); // TPL.FB_MODULECONTROLLER
iq_stStandardModuleItf.q_xActive := fbModuleController.q_xActive;

// NETWORK 2
// Distributes jogging Inputs to all Axis modules
//   iq_stStandardModuleItf.i_xEnable: stI : ST_StandardModuleInterfaceIn;
//   iq_stStandardModuleItf: TPL.ST_StandardModuleInterface
//   iq_stStandardMotionItf: TPL.ST_StandardMotionInterface
//   iq_stExceptionList: ExceptionHandling and Logging
fbAxisModuleController(
    i_xEnable := iq_stStandardModuleItf.i_xEnable,
    iq_stStandardModuleItf := iq_stStandardModuleItf,
    iq_stStandardMotionItf := iq_stStandardMotionItf,
    iq_stExceptionList := iq_stExceptionList,
    iq_stLogDataList := iq_stLogDataList); // AXM.FB_AXISMODULECONTROLLER

// NETWORK 3
// (* End of system generated code, could be modified for your application *)
//   iq_stExceptionList: ExceptionHandling and Logging
//   stMasterInterface: User specific variables
fbMasterModule(
    iq_stStandardModuleItf := astSubModuleInterface[c_udiMaster],
    iq_stExceptionList := iq_stExceptionList,
    iq_stLogDataList := iq_stLogDataList,
    iq_stAxisModuleItf := stMasterInterface); // AXM.FB_AXISMODULE
END_ACTION

ACTION UpdateStructs:
(* System generated code, do not change without consulting 'Schneider Electric Automation GmbH' - otherwise you risk instability!!! *)
fbDetectOnlineChange(	i_xEnable	:= TRUE, 
						i_xDetect	:= TRUE, 
						q_xActive	=> xDetectOnlineChangeActive, 
						q_xReady	=> xDetectOnlineChangeReady, 
						q_etDiag	=> etDetectOnlineChangeDiag, 
						q_etDiagExt	=> etDetectOnlineChangeDiagExt, 
						q_sMsg		=> sDetectOnlineChangeMsg, 
						q_xChange	=> );
						
IF(NOT fbDetectOnlineChange.q_xChange) THEN
	RETURN;
END_IF

iq_stStandardModuleItf.iq_stExt.udiNumberOfSubModules 		:= c_udiNumberOfSubModules;
iq_stStandardModuleItf.iq_stExt.dwSubModulesItf		 		:= ADR(astSubModuleInterface);
iq_stStandardModuleItf.iq_stExt.pdwSubModulesAddItf		 	:= ADR(adwSubModuleAddInterfaces);
iq_stStandardModuleItf.iq_stExt.pstListOfCmdTables			:= ADR(astListOfCmdTables);
iq_stStandardModuleItf.iq_stExt.udiNumberOfCmdTables		:= c_udiNumberOfCmdTables;
(* End of system generated code, do not change without consulting 'Schneider Electric Automation GmbH' - otherwise you risk instability!!! *)

(* System generated code, could be modified for your application *)
xUpdateStructsException := FALSE;

(*****************************************************************************************************************************************************)
(* Update CmdTable - Prepare *)

TPL.FC_UpdateCmdTableListElement(	i_pstListofCmdTables	:= ADR(astListOfCmdTables),
									i_udiNumberOfCmdTables	:= c_udiNumberOfCmdTables,
									i_diCmd					:= ET_Cmd.Prepare,
									i_pstCmdTable			:= ADR(astPrepareTable),
									q_etDiag				=> etDiag,
									q_etDiagExt				=> etDiagExtTPL);
									
IF etDiag <> GD.ET_Diag.Ok AND NOT xUpdateStructsException THEN
	xUpdateStructsException := TRUE;
	
	stUpdateStructsException.sMsg := PDL.FC_MultiConcat(i_sString1 := 'Update CmdTable: Prepare - ', 
														i_sString2 := GD.FC_EtDiagToString(i_etDiag := etDiag), 
														i_sString3 := ' - ', 
														i_sString4 := TPL.FC_EtDiagExtToString(i_etDiagExt := etDiagExtTPL));
END_IF										

(*****************************************************************************************************************************************************)
(* Update CmdTable - Auto *)

TPL.FC_UpdateCmdTableListElement(	i_pstListofCmdTables	:= ADR(astListOfCmdTables),
									i_udiNumberOfCmdTables	:= c_udiNumberOfCmdTables,
									i_diCmd					:= ET_Cmd.Auto,
									i_pstCmdTable			:= ADR(astAutoTable),
									q_etDiag				=> etDiag,
									q_etDiagExt				=> etDiagExtTPL);
									
IF etDiag <> GD.ET_Diag.Ok AND NOT xUpdateStructsException THEN
	xUpdateStructsException := TRUE;
	
	stUpdateStructsException.sMsg := PDL.FC_MultiConcat(i_sString1 := 'Update CmdTable: Auto - ', 
														i_sString2 := GD.FC_EtDiagToString(i_etDiag := etDiag), 
														i_sString3 := ' - ', 
														i_sString4 := TPL.FC_EtDiagExtToString(i_etDiagExt := etDiagExtTPL));
END_IF		

(*****************************************************************************************************************************************************)
(* Update CmdTable - Manual *)

TPL.FC_UpdateCmdTableListElement(	i_pstListofCMDTables	:= ADR(astListofCMDTables),
									i_udiNumberOfCMDTables	:= c_udiNumberOfCMDTables,
									i_diCMD					:= ET_Cmd.Manual,
									i_pstCMDTable			:= ADR(astManualTable),
									q_etDiag				=> etDiag,
									q_etDiagExt				=> etDiagExtTPL);
									
IF etDiag <> GD.ET_Diag.Ok AND NOT xUpdateStructsException THEN
	xUpdateStructsException := TRUE;
	
	stUpdateStructsException.sMsg := PDL.FC_MultiConcat(i_sString1 := 'Update CmdTable: Manual - ', 
														i_sString2 := GD.FC_EtDiagToString(i_etDiag := etDiag), 
														i_sString3 := ' - ', 
														i_sString4 := TPL.FC_EtDiagExtToString(i_etDiagExt := etDiagExtTPL));
END_IF		

(*****************************************************************************************************************************************************)
(* Update CmdTable - Stop *)

TPL.FC_UpdateCmdTableListElement(	i_pstListofCMDTables	:= ADR(astListofCMDTables),
									i_udiNumberOfCMDTables	:= c_udiNumberOfCMDTables,
									i_diCMD					:= ET_Cmd.Stop,
									i_pstCMDTable			:= ADR(astStopTable),
									q_etDiag				=> etDiag,
									q_etDiagExt				=> etDiagExtTPL);
									
IF etDiag <> GD.ET_Diag.Ok AND NOT xUpdateStructsException THEN
	xUpdateStructsException := TRUE;
	
	stUpdateStructsException.sMsg := PDL.FC_MultiConcat(i_sString1 := 'Update CmdTable: Stop - ', 
														i_sString2 := GD.FC_EtDiagToString(i_etDiag := etDiag), 
														i_sString3 := ' - ', 
														i_sString4 := TPL.FC_EtDiagExtToString(i_etDiagExt := etDiagExtTPL));
END_IF		

(*****************************************************************************************************************************************************)
(* Update CmdTable - Start *)

TPL.FC_UpdateCmdTableListElement(	i_pstListofCMDTables	:= ADR(astListofCMDTables),
									i_udiNumberOfCmdTables	:= c_udiNumberOfCMDTables,
									i_diCMD					:= ET_Cmd.Start,
									i_pstCMDTable			:= ADR(astStartTable),
									q_etDiag				=> etDiag,
									q_etDiagExt				=> etDiagExtTPL);
									
IF etDiag <> GD.ET_Diag.Ok AND NOT xUpdateStructsException THEN
	xUpdateStructsException := TRUE;
	
	stUpdateStructsException.sMsg := PDL.FC_MultiConcat(i_sString1 := 'Update CmdTable: Start - ', 
														i_sString2 := GD.FC_EtDiagToString(i_etDiag := etDiag), 
														i_sString3 := ' - ', 
														i_sString4 := TPL.FC_EtDiagExtToString(i_etDiagExt := etDiagExtTPL));
END_IF		

(*****************************************************************************************************************************************************)
(* Update CmdTable - Abort *)

TPL.FC_UpdateCmdTableListElement(	i_pstListofCMDTables	:= ADR(astListofCMDTables),
									i_udiNumberOfCmdTables	:= c_udiNumberOfCmdTables,
									i_diCMD					:= ET_Cmd.Abort,
									i_pstCMDTable			:= ADR(astAbortTable),
									q_etDiag				=> etDiag,
									q_etDiagExt				=> etDiagExtTPL);
									
IF etDiag <> GD.ET_Diag.Ok AND NOT xUpdateStructsException THEN
	xUpdateStructsException := TRUE;
	
	stUpdateStructsException.sMsg := PDL.FC_MultiConcat(i_sString1 := 'Update CmdTable: Abort - ', 
														i_sString2 := GD.FC_EtDiagToString(i_etDiag := etDiag), 
														i_sString3 := ' - ', 
														i_sString4 := TPL.FC_EtDiagExtToString(i_etDiagExt := etDiagExtTPL));
END_IF		

(*****************************************************************************************************************************************************)
(* Update CmdTable - Hold *)

TPL.FC_UpdateCmdTableListElement(	i_pstListofCMDTables	:= ADR(astListofCMDTables),
									i_udiNumberOfCmdTables	:= c_udiNumberOfCmdTables,
									i_diCMD					:= ET_Cmd.Hold,
									i_pstCMDTable			:= ADR(astHoldTable),
									q_etDiag				=> etDiag,
									q_etDiagExt				=> etDiagExtTPL);
									
IF etDiag <> GD.ET_Diag.Ok AND NOT xUpdateStructsException THEN
	xUpdateStructsException := TRUE;
	
	stUpdateStructsException.sMsg := PDL.FC_MultiConcat(i_sString1 := 'Update CmdTable: Hold - ', 
														i_sString2 := GD.FC_EtDiagToString(i_etDiag := etDiag), 
														i_sString3 := ' - ', 
														i_sString4 := TPL.FC_EtDiagExtToString(i_etDiagExt := etDiagExtTPL));
END_IF		

(*****************************************************************************************************************************************************)
(* Update CmdTable - BrakeRelease *)

TPL.FC_UpdateCmdTableListElement(	i_pstListofCMDTables	:= ADR(astListofCMDTables),
									i_udiNumberOfCMDTables	:= c_udiNumberOfCMDTables,
									i_diCMD					:= ET_Cmd.BrakeRelease,
									i_pstCMDTable			:= ADR(astBrakeReleaseTable),
									q_etDiag				=> etDiag,
									q_etDiagExt				=> etDiagExtTPL);
									
IF etDiag <> GD.ET_Diag.Ok AND NOT xUpdateStructsException THEN
	xUpdateStructsException := TRUE;
	
	stUpdateStructsException.sMsg := PDL.FC_MultiConcat(i_sString1 := 'Update CmdTable: BrakeRelease - ', 
														i_sString2 := GD.FC_EtDiagToString(i_etDiag := etDiag), 
														i_sString3 := ' - ', 
														i_sString4 := TPL.FC_EtDiagExtToString(i_etDiagExt := etDiagExtTPL));
END_IF		
									
(*****************************************************************************************************************************************************)
(* Update AddInterface - Master *)

AXM.FC_UpdateAddInterfaceStruct(	i_pdwSubModuleAddInterfaces	:= ADR(adwSubModuleAddInterfaces),
									i_udiSubModuleConstant		:= c_udiMaster,
									iq_stAxisModuleItf			:= stMasterInterface,
									q_etDiag					=> etDiag,
									q_etDiagExt					=> etDiagExtAXM);
									
IF etDiag <> GD.ET_Diag.Ok AND NOT xUpdateStructsException THEN
	xUpdateStructsException := TRUE;
	
	stUpdateStructsException.sMsg := PDL.FC_MultiConcat(i_sString1 := 'Update AddInterface: Master - ', 
														i_sString2 := GD.FC_EtDiagToString(i_etDiag := etDiag), 
														i_sString3 := ' - ', 
														i_sString4 := AXM.FC_EtDiagExtToString(i_etDiagExt := etDiagExtAXM));
END_IF		

(*****************************************************************************************************************************************************)
(* Update ILS Data *)

// stMasterInterface.stEndless.pstIlsData	:= ADR(G_stIlsData);
// stMasterInterface.stMultiCam.pstIlsData	:= ADR(G_stIlsData);

(*****************************************************************************************************************************************************)
(* Set exception if any exception occurred *)

